	            // ss_SequencialID character string leading zeros addition
	            IF (#si_StringLen < 6)
	            THEN
	                FOR #si_LenFillLoop := 1 TO 6 - #si_StringLen DO
	                    #ss_SequencialID := CONCAT(IN1 := '0',
	                                               IN2 := #ss_SequencialID);
	                END_FOR;
	            END_IF;
	        END_REGION

	        REGION 3.2 LLC Syatem ID
	            // Build LLC Syatem ID
	            #ss_LLCSystemID := CONCAT(IN1 := #is_DEPCOD,
	                                      IN2 := #is_LOConEquipment,
	                                      IN3 := #is_TYPofEquipment,
	                                      IN4 := #is_NumberOfTheEquipment);

	        END_REGION

	        REGION 3.3 - Package ID
	            // Build Package ID
	            #ss_PackageID := CONCAT(IN1 := #is_TrayCellNumber,
	                                    IN2 := #is_SorterNumber,
	                                    IN3 := #is_InductionNumber,
	                                    IN4 := #is_AreaNumber,
	                                    IN5 := #ss_SequencialID);
	        END_REGION

	        REGION 3.4 - Gap

	            // Gap character string clearing
	            #ss_Gap := '';

	            IF ("DB_GIN".GIN[#ii_Gin].General.LeadingGap > 999)
	            THEN
	                #ss_Gap := '999';
	            ELSE

	                // Gap integer input conversion to a character string
	                VAL_STRG(IN := "DB_GIN".GIN[#ii_Gin].General.LeadingGap,
	                         SIZE := 0,
	                         PREC := 0,
	                         FORMAT := 0,
	                         P := 1,
	                         OUT => #ss_Gap);
	                // Length of the gap character string
	                #si_StringLen := LEN(#ss_Gap);
	                // Gap character string leading zeros addition
	                IF (#si_StringLen < 3)
	                THEN
	                    FOR #si_LenFillLoop := 1 TO 3 - #si_StringLen DO
	                        #ss_Gap := CONCAT(IN1 := '0',
	                                          IN2 := #ss_Gap);
	                    END_FOR;
	                END_IF;

	            END_IF;

	        END_REGION

	        REGION 3.5 – Message preparation

	            // Message composing according to the structure: STX,message body,ETX
	            #ss_MessageP1 := CONCAT(IN1 := #cc_STX,
	                                    IN2 := #cs_Length,
	                                    IN3 := #cs_MessageType,
	                                    IN4 := #ss_LLCSystemID,
	                                    IN5 := "DB_GIN".GIN[#ii_Gin].FedEx.ADCSystemID,
	                                    IN6 := "DB_GIN".GIN[#ii_Gin].FedEx.ImageID,
	                                    IN7 := #ss_PackageID,
	                                    IN8 := "DB_GIN".GIN[#ii_Gin].FedEx.HLCPackageID,
	                                    IN9 := "DB_GIN".GIN[#ii_Gin].FedEx.DIMSystemID,
	                                    IN10 := "DB_GIN".GIN[#ii_Gin].FedEx.DIMStatus,
	                                    IN11 := "DB_GIN".GIN[#ii_Gin].FedEx.PackageDimLength,
	                                    IN12 := "DB_GIN".GIN[#ii_Gin].FedEx.PackageDimWidth,
	                                    IN13 := "DB_GIN".GIN[#ii_Gin].FedEx.PackageDimHeight,
	                                    IN14 := #ss_Gap,
	                                    IN15 := "DB_GIN".GIN[#ii_Gin].FedEx.DIMUOM,
	                                    IN16 := "DB_GIN".GIN[#ii_Gin].FedEx.DimLFTstatusCode,
	                                    IN17 := "DB_GIN".GIN[#ii_Gin].FedEx.AlibiDims,
	                                    IN18 := "DB_GIN".GIN[#ii_Gin].FedEx.SCLSystemID,
	                                    IN19 := "DB_GIN".GIN[#ii_Gin].FedEx.SCLWT,
	                                    IN20 := "DB_GIN".GIN[#ii_Gin].FedEx.SCLWTUOM,
	                                    IN21 := "DB_GIN".GIN[#ii_Gin].FedEx.SCLLFTStatusCode,
	                                    IN22 := "DB_GIN".GIN[#ii_Gin].FedEx.AlibiWeight,
	                                    IN23 := "DB_GIN".GIN[#ii_Gin].FedEx.ReasonCode,
	                                    IN24 := "DB_Time".Timestamp,
	                                    IN25 := #iUDT_Facility.TimeZoneDesignator);

	            #ss_MessageP2 := CONCAT(IN1 := "DB_GIN".GIN[#ii_Gin].FedEx.Barcode1Identification,
	                                    IN2 := "DB_GIN".GIN[#ii_Gin].FedEx.Barcode1status,
	                                    IN3 := "DB_GIN".GIN[#ii_Gin].FedEx.Barcode1datalength,
	                                    IN4 := "DB_GIN".GIN[#ii_Gin].FedEx.Barcode1data,
	                                    IN5 := #cc_ETX);

	        END_REGION

	        REGION 3.6 – Maximum number of the message characters

	            #si_MaxMsgLen := "FC_GetNrOfArrayEl"(iv_Array := #sUDT_MessageArray.Character);

	        END_REGION

	        REGION 3.7 – Length of the complete message

	            #si_MsgLen := LEN(#ss_MessageP1) + LEN(#ss_MessageP2);
	            // Message length validation
	            #sa_Status.InvalidMessageLength := #si_MsgLen - 2 <> STRING_TO_INT(#cs_Length);

	        END_REGION

	        REGION 3.8 –  Message array size validation

	            #sa_Status.InvalidMsgArraySize := #si_MsgLen > #si_MaxMsgLen;

	        END_REGION

	        REGION 3.9 –  Message character string conversion to a message array of characters

	            IF (NOT #sa_Status.InvalidMsgArraySize)     // Message character array size is valid
	            THEN

	                Strg_TO_Chars(Strg := #ss_MessageP1,
	                              pChars := 0,
	                              Cnt => #sui_ArrayOffset,
	                              Chars := #sUDT_MessageArray.Character);

	                Strg_TO_Chars(Strg := #ss_MessageP2,
	                              pChars := #sui_ArrayOffset,
	                              Cnt => #sui_MsgArrayElNr,
	                              Chars := #sUDT_MessageArray.Character);

	            END_IF;

	        END_REGION

	        REGION 3.10 – Clearing remaining characters in the message character array

	            IF (NOT #sa_Status.InvalidMsgArraySize)     // Message character array size is valid
	            THEN

	                // Filling up not used message character array elements with '$00' (ASCII - 16#00)
	                FILL_BLK(IN := #cc_NULL,                                                                             // Fill not used message char array elements with '$00'
	                         COUNT := UINT_TO_ULINT(INT_TO_UINT(#si_MaxMsgLen) - #sui_MsgArrayElNr - #sui_ArrayOffset),
	                         OUT => #sUDT_MessageArray.Character[#sui_MsgArrayElNr + #sui_ArrayOffset]);

	            END_IF;

	        END_REGION

	        REGION 3.11 – Message write into a FIFO register

	            IF NOT #sa_Status.InvalidMsgArraySize               // Message character array size is valid
	                AND NOT #sa_Status.InvalidMessageLength         //Message length is valid
	            THEN

	                // Mode 'W' - Write FIFO record
	                "FC_Fifo"(ic_Mode := 'W',
	                          qUDT_Status => #sa_Status.FIFOStatus,
	                          qx_Error => #sa_Status.FIFOError,
	                          qx_Warning => #sa_Status.FIFOWarning,
	                          iqv_Data := #sUDT_MessageArray,
	                          iqUDT_FifoHeader := #iqUDT_FifoHeader,
	                          iqv_DataBuffer := #iqa_FifoData);
	            ELSE
	                // Increase counter messages not sent because of wrong message length
	                #sa_Statistics.NotSentWrongMsgLen += 1;

	            END_IF;

	            #si_OldGin := #ii_Gin;
	        END_REGION


	        // In case of FIFO full, the FIFO full error bit and FIFO collective error bit are set
	    ELSE
	        #sa_Status.FIFOError := TRUE;
	        #sa_Status.FIFOStatus.FifoFull := TRUE;
	    END_IF;



	END_REGION

	REGION 4 - Writing outputs

	    #sx_Error := #sa_Status.InvalidMessageLength        // Invalid message length
	    OR #sa_Status.InvalidGIN                            // Invalid GIN
	    OR #sa_Status.InvalidMsgArraySize                   // Invalid message array size
	    OR #sa_Status.FIFOError;                            // FIFO error

	END_REGION



	REGION 5 Unexpected DX Request

	    IF #iqx_Unexpected_DX_Req THEN

	        REGION 5.1 – FIFO header status update

	            // Mode 'S' - FIFO register status update
	            "FC_Fifo"(ic_Mode := 'S',
	                      qUDT_Status => #sa_Status.FIFOStatus,
	                      qx_Error => #sa_Status.FIFOError,
	                      qx_Warning => #sa_Status.FIFOWarning,
	                      iqv_Data := #sUDT_MessageArray,
	                      iqUDT_FifoHeader := #iqUDT_FifoHeader,
	                      iqv_DataBuffer := #iqa_FifoData);
	        END_REGION

	        REGION 5.2 – Message preparation

	            IF NOT #iqUDT_FifoHeader.Status.Full       // FIFO isn't full
	            THEN
	                REGION Sequencial ID
	                    // ss_SequencialID character string clearing
	                    #ss_SequencialID := '';
	                    // ss_SequencialID integer input conversion to a character string
	                    VAL_STRG(IN := "DB_ExternalGIN".UnexpectedSI.FedEx.CustomerID,
	                             SIZE := 0,
	                             PREC := 0,
	                             FORMAT := 0,
	                             P := 1,
	                             OUT => #ss_SequencialID);
	                    // Length of the ss_SequencialID character string
	                    #si_StringLen := LEN(#ss_SequencialID);

	                    // ss_SequencialID character string leading zeros addition
	                    IF (#si_StringLen < 6)
	                    THEN
	                        FOR #si_LenFillLoop := 1 TO 6 - #si_StringLen DO
	                            #ss_SequencialID := CONCAT(IN1 := '0',
	                                                       IN2 := #ss_SequencialID);
	                        END_FOR;
	                    END_IF;
	                END_REGION

	                REGION LLC Syatem ID
	                    // Build LLC Syatem ID
	                    #ss_LLCSystemID := CONCAT(IN1 := #is_DEPCOD,
	                                              IN2 := #is_LOConEquipment,
	                                              IN3 := #is_TYPofEquipment,
	                                              IN4 := #is_NumberOfTheEquipment);

	                END_REGION

	                REGION Package ID
	                    // Build Package ID
	                    #ss_PackageID := CONCAT(IN1 := #is_TrayCellNumber,
	                                            IN2 := #is_SorterNumber,
	                                            IN3 := #is_InductionNumber,
	                                            IN4 := #is_AreaNumber,
	                                            IN5 := #ss_SequencialID);
	                END_REGION

	                REGION Gap

	                    #ss_Gap := '000';

	                END_REGION

	                REGION 3.5 – Message preparation

	                    // Message composing according to the structure: STX,message body,ETX
	                    #ss_MessageP1 := CONCAT(IN1 := #cc_STX,
	                                            IN2 := #cs_Length,
	                                            IN3 := #cs_MessageType,
	                                            IN4 := #ss_LLCSystemID,
	                                            IN5 := "DB_ExternalGIN".UnexpectedSI.FedEx.ADCSystemID,
	                                            IN6 := "DB_ExternalGIN".UnexpectedSI.FedEx.ImageID,
	                                            IN7 := "DB_ExternalGIN".UnexpectedSI.FedEx.PackageID,
	                                            IN8 := "DB_ExternalGIN".UnexpectedSI.FedEx.HLCPackageID,
	                                            IN9 := "DB_ExternalGIN".UnexpectedSI.FedEx.DIMSystemID,
	                                            IN10 := "DB_ExternalGIN".UnexpectedSI.FedEx.DIMStatus,
	                                            IN11 := "DB_ExternalGIN".UnexpectedSI.FedEx.PackageDimLength,
	                                            IN12 := "DB_ExternalGIN".UnexpectedSI.FedEx.PackageDimWidth,
	                                            IN13 := "DB_ExternalGIN".UnexpectedSI.FedEx.PackageDimHeight,
	                                            IN14 := #ss_Gap,
	                                            IN15 := "DB_ExternalGIN".UnexpectedSI.FedEx.DIMUOM,
	                                            IN16 := "DB_ExternalGIN".UnexpectedSI.FedEx.DimLFTstatusCode,
	                                            IN17 := "DB_ExternalGIN".UnexpectedSI.FedEx.AlibiDims,
	                                            IN18 := "DB_ExternalGIN".UnexpectedSI.FedEx.SCLSystemID,
	                                            IN19 := "DB_ExternalGIN".UnexpectedSI.FedEx.SCLWT,
	                                            IN20 := "DB_ExternalGIN".UnexpectedSI.FedEx.SCLWTUOM,
	                                            IN21 := "DB_ExternalGIN".UnexpectedSI.FedEx.SCLLFTStatusCode,
	                                            IN22 := "DB_ExternalGIN".UnexpectedSI.FedEx.AlibiWeight,
	                                            IN23 := "DB_ExternalGIN".UnexpectedSI.FedEx.ReasonCode,
	                                            IN24 := "DB_Time".Timestamp,
	                                            IN25 := #iUDT_Facility.TimeZoneDesignator);

	                    #ss_MessageP2 := CONCAT(IN1 := "DB_ExternalGIN".UnexpectedSI.FedEx.Barcode1Identification,
	                                            IN2 := "DB_ExternalGIN".UnexpectedSI.FedEx.Barcode1status,
	                                            IN3 := "DB_ExternalGIN".UnexpectedSI.FedEx.Barcode1datalength,
	                                            IN4 := "DB_ExternalGIN".UnexpectedSI.FedEx.Barcode1data,
	                                            IN5 := #cc_ETX);

	                END_REGION

	                REGION 3.6 – Maximum number of the message characters

	                    #si_MaxMsgLen := "FC_GetNrOfArrayEl"(iv_Array := #sUDT_MessageArray.Character);

	                END_REGION

	                REGION 3.7 – Length of the complete message

	                    #si_MsgLen := LEN(#ss_MessageP1) + LEN(#ss_MessageP2);
	                    // Message length validation
	                    #sa_Status.InvalidMessageLength := #si_MsgLen - 2 <> STRING_TO_INT(#cs_Length);

	                END_REGION

	                REGION 3.8 –  Message array size validation

	                    #sa_Status.InvalidMsgArraySize := #si_MsgLen > #si_MaxMsgLen;

	                END_REGION

	                REGION 3.9 –  Message character string conversion to a message array of characters

	                    IF (NOT #sa_Status.InvalidMsgArraySize)     // Message character array size is valid
	                    THEN

	                        Strg_TO_Chars(Strg := #ss_MessageP1,
	                                      pChars := 0,
	                                      Cnt => #sui_ArrayOffset,
	                                      Chars := #sUDT_MessageArray.Character);

	                        Strg_TO_Chars(Strg := #ss_MessageP2,
	                                      pChars := #sui_ArrayOffset,
	                                      Cnt => #sui_MsgArrayElNr,
	                                      Chars := #sUDT_MessageArray.Character);

	                    END_IF;

	                END_REGION

	                REGION 3.10 – Clearing remaining characters in the message character array

	                    IF (NOT #sa_Status.InvalidMsgArraySize)     // Message character array size is valid
	                    THEN

	                        // Filling up not used message character array elements with '$00' (ASCII - 16#00)
	                        FILL_BLK(IN := #cc_NULL,                                                                             // Fill not used message char array elements with '$00'
	                                 COUNT := UINT_TO_ULINT(INT_TO_UINT(#si_MaxMsgLen) - #sui_MsgArrayElNr - #sui_ArrayOffset),
	                                 OUT => #sUDT_MessageArray.Character[#sui_MsgArrayElNr + #sui_ArrayOffset]);

	                    END_IF;

	                END_REGION

	                REGION 3.11 – Message write into a FIFO register

	                    IF NOT #sa_Status.InvalidMsgArraySize               // Message character array size is valid
	                        AND NOT #sa_Status.InvalidMessageLength         //Message length is valid
	                    THEN

	                        // Mode 'W' - Write FIFO record
	                        "FC_Fifo"(ic_Mode := 'W',
	                                  qUDT_Status => #sa_Status.FIFOStatus,
	                                  qx_Error => #sa_Status.FIFOError,
	                                  qx_Warning => #sa_Status.FIFOWarning,
	                                  iqv_Data := #sUDT_MessageArray,
	                                  iqUDT_FifoHeader := #iqUDT_FifoHeader,
	                                  iqv_DataBuffer := #iqa_FifoData);
	                    ELSE
	                        // Increase counter messages not sent because of wrong message length
	                        #sa_Statistics.NotSentWrongMsgLen += 1;

	                    END_IF;

	                END_REGION
	                #iqx_Unexpected_DX_Req := FALSE;


	                // In case of FIFO full, the FIFO full error bit and FIFO collective error bit are set
	            ELSE
	                #sa_Status.FIFOError := TRUE;
	                #sa_Status.FIFOStatus.FifoFull := TRUE;
	            END_IF;

	        END_REGION
	    END_IF;
	END_REGION



	REGION 6 - Writing outputs

	    #qx_Error := #sa_Status.InvalidMessageLength        // Invalid message length
	    OR #sa_Status.InvalidGIN                            // Invalid GIN
	    OR #sa_Status.InvalidMsgArraySize                   // Invalid message array size
	    OR #sa_Status.FIFOError                             // FIFO error
	    OR #sx_Error;

	END_REGION
END_FUNCTION_BLOCK

FUNCTION_BLOCK "FB_FedExEntrancePoint"
{ S7_Optimized_Access := 'TRUE' }
VERSION : 0.1
// ATTRIBUTES
// AUTO_NUMBER = True
// BLOCK_NUMBER = 71
// END_ATTRIBUTES
   VAR_INPUT
      is_PackageEntrancePoint { ExternalAccessible := 'False'; ExternalVisible := 'False'; ExternalWritable := 'False'} : String;
      is_PackageEntranceState { ExternalAccessible := 'False'; ExternalVisible := 'False'; ExternalWritable := 'False'} : String;
      ii_Gin { ExternalAccessible := 'False'; ExternalVisible := 'False'; ExternalWritable := 'False'} : Int;
   END_VAR

   VAR
      si_OldGIN { ExternalAccessible := 'False'; ExternalVisible := 'False'; ExternalWritable := 'False'} : Int;
      si_StringLen { ExternalAccessible := 'False'; ExternalVisible := 'False'; ExternalWritable := 'False'} : Int;
      si_LenFillLoop { ExternalAccessible := 'False'; ExternalVisible := 'False'; ExternalWritable := 'False'} : Int;
   END_VAR

   VAR_TEMP
      tx_InvalidGIN : Bool;
   END_VAR


BEGIN
	(*
	----------------------------------------------------------------------------------------

	Version history:
	Date        | Version   | Author        | Remark
	----------------------------------------------------------------------------------------
	30/06/2022  | 0.1       | K. Pokorski   | first release MHS TIA 16
	21/02/2023  | 4.0       | F.Baten       | 4.0 Release TIA 17.5
	*)

	REGION 1 - GIN validation

	    // GIN validation
	    #tx_InvalidGIN := (#ii_Gin < 1) OR (#ii_Gin > 9999);

	    IF #ii_Gin <> #si_OldGIN AND NOT #tx_InvalidGIN
	    THEN

	        "DB_GIN".GIN[#ii_Gin].FedEx.PackageEntrancePoint := #is_PackageEntrancePoint;
	        "DB_GIN".GIN[#ii_Gin].FedEx.PackageEntranceState := #is_PackageEntranceState;

	        #si_StringLen := LEN("DB_GIN".GIN[#ii_Gin].FedEx.PackageEntrancePoint);

	        IF (#si_StringLen < 14)
	        THEN
	            FOR #si_LenFillLoop := 1 TO 14 - #si_StringLen DO

	                "DB_GIN".GIN[#ii_Gin].FedEx.PackageEntrancePoint := CONCAT(IN1 := "DB_GIN".GIN[#ii_Gin].FedEx.PackageEntrancePoint,
	                                                                           IN2 := ' ');
	            END_FOR;
	        END_IF;

	        #si_OldGIN := #ii_Gin;

	    END_IF;


	END_REGION






END_FUNCTION_BLOCK

FUNCTION_BLOCK "FB_FedExGetPositionPolisorter"
TITLE = FB_GetPosition
{ S7_Optimized_Access := 'TRUE' }
FAMILY : MHS
VERSION : 3.0
// ATTRIBUTES
// AUTO_NUMBER = True
// BLOCK_NUMBER = 73
// END_ATTRIBUTES
//Function to find the position based on the GIN in the tracking.
   VAR_INPUT
      idi_ConveyorLength { ExternalAccessible := 'False'; ExternalVisible := 'False'; ExternalWritable := 'False'} : DInt;   // Conveyor length [mm]
      idi_WaitDistanceCorrection { ExternalAccessible := 'False'; ExternalVisible := 'False'; ExternalWritable := 'False'} : DInt := 10000;   // Distance how much parcel tail can stick out of the conveyor [mm]
   END_VAR

   VAR_IN_OUT
      iqs_DBDestination : Array[*] of "UDT_FedExDestinations";   // Array with destination data for parcel
      iqUDT_PolisorterInterface : "UDT_PolisorterInterface";   // Interface beween VSU and VFD
      iqUDT_ConveyorInterface : "UDT_ConveyorInterface";   // Polisorter conveyor interface structure
      iqs_TrackingData : Array[*] of Int;   // Tracking data
   END_VAR

   VAR
      si_Gin { ExternalAccessible := 'False'; ExternalVisible := 'False'; ExternalWritable := 'False'} : Int;   // GIN
      si_PreviousGin { ExternalAccessible := 'False'; ExternalVisible := 'False'; ExternalWritable := 'False'} : Int;   // Old GIN memeory
      si_RequestedDestination { ExternalAccessible := 'False'; ExternalVisible := 'False'; ExternalWritable := 'False'} : Int;   // The destination for this GIN
      si_RequestedPosition { ExternalAccessible := 'False'; ExternalVisible := 'False'; ExternalWritable := 'False'} : Int;   // Requested position
      si_LC_Positions { ExternalAccessible := 'False'; ExternalVisible := 'False'; ExternalWritable := 'False'} : Int;   // Loopcounter positions
      si_LC_Destinations { ExternalAccessible := 'False'; ExternalVisible := 'False'; ExternalWritable := 'False'} : Int;   // Loopcounter destinations
      si_NrPositons { ExternalAccessible := 'False'; ExternalVisible := 'False'; ExternalWritable := 'False'} : Int;   // Number of positions in the search area
      si_NrDestinations { ExternalAccessible := 'False'; ExternalVisible := 'False'; ExternalWritable := 'False'} : Int;   // Number of destinations per position
      sx_NewGinFound { ExternalAccessible := 'False'; ExternalVisible := 'False'; ExternalWritable := 'False'} : Bool;   // Memory to start searching
      sdi_WaitDistance { ExternalAccessible := 'False'; ExternalVisible := 'False'; ExternalWritable := 'False'} : DInt;   // Calculated wait distance [cm]
      sdi_ParcelLength { ExternalAccessible := 'False'; ExternalVisible := 'False'; ExternalWritable := 'False'} : DInt;   // Parcel length [cm]
   END_VAR


BEGIN
	(*
	----------------------------------------------------------------------------------------
	|                                                                                      |
	|  Copyright  2019             MHS                                                     |
	|  All Rights Reserved         Larenweg 90                                             |
	|                              5234 KC 's-Hertogenbosch,                               |
	|                              Netherlands                                             |
	|                                                                                      |
	----------------------------------------------------------------------------------------

	Version history:
	Date        | Version   | Author        | Remark
	----------------------------------------------------------------------------------------

	26/01/2022  | 0.1       | L.Klar        | Initial version
	13/03/2024  | 4.1       | S. Nieświec   | 4.1 Release TIA 18
	02/05/2024  | 4.2       | J.Majer      | Datatype conversions changed from automatic to explicit, to accomodate IEC 61131-3 standard
	*)

	REGION 1 - Determine size of search area

	    #si_NrPositons := "FC_GetNrOfArrayEl"(#iqs_DBDestination);
	    #si_NrDestinations := "FC_GetNrOfArrayEl"(#iqs_DBDestination[1].Destination);

	END_REGION

	REGION 2 - Get GIN from tracking DB

	    // There is a value in the tracking data on the decision point which is not '0' or equal to the previous GIN
	    IF (#iqs_TrackingData[#iqUDT_PolisorterInterface.Decisionpoint] <> 0) AND (#iqs_TrackingData[#iqUDT_PolisorterInterface.Decisionpoint] <> #si_PreviousGin)
	    THEN
	        #si_Gin := #iqs_TrackingData[#iqUDT_PolisorterInterface.Decisionpoint];
	        #sx_NewGinFound := TRUE;
	    END_IF;

	END_REGION

	REGION 3 - Wait distance

	    IF #sdi_WaitDistance > 0 THEN
	        #sdi_WaitDistance -= #iqUDT_ConveyorInterface.Displacement;
	    END_IF;

	END_REGION

	REGION 4 - Get destination from GIN DB
	    // If new GIN has been detected, get destination from its GIN record

	    IF #sx_NewGinFound AND #si_Gin > 0
	    THEN
	        #si_RequestedDestination := DINT_TO_INT("DB_GIN".GIN[#si_Gin].General.Destination[0]);

	        #sdi_ParcelLength := "DB_GIN".GIN[#si_Gin].General.Length;

	        // If parcel length is lower than conveyor length - decision point use calculated decision point to switch.
	        // If not, then caluclate additional wait distance, based on correction factor
	        // If the parcel length is equal to 0, use fixed wait distance of decision point minus 40
	        IF #sdi_ParcelLength > 0
	        THEN
	            IF #sdi_ParcelLength < #idi_ConveyorLength / 10 - #iqUDT_PolisorterInterface.Decisionpoint
	            THEN
	                #sdi_WaitDistance := 0;
	            ELSE
	                #sdi_WaitDistance := #sdi_ParcelLength - (#idi_ConveyorLength / 10 - #iqUDT_PolisorterInterface.Decisionpoint) - #idi_WaitDistanceCorrection / 10;
	            END_IF;
	        ELSE
	            #sdi_WaitDistance := #iqUDT_PolisorterInterface.Decisionpoint - 40;
	        END_IF;
	        #si_PreviousGin := #si_Gin;
	        #si_Gin := 0;
	        #iqUDT_PolisorterInterface.RequestedPosition := 0;

	    END_IF;

	END_REGION

	REGION 5 - Get requested position when new GIN is found

	    IF #sx_NewGinFound AND #sdi_WaitDistance <= 0
	    THEN
	        // If destination is different than 0, find a position in destination arrays. Otherwise, requested position is set to default.
	        IF #si_RequestedDestination <> 0 THEN
	            FOR #si_LC_Positions := 1 TO #si_NrPositons BY 1 DO
	                FOR #si_LC_Destinations := 0 TO (#si_NrDestinations - 1) BY 1 DO
	                    IF #iqs_DBDestination[#si_LC_Positions].Destination[#si_LC_Destinations] = #si_RequestedDestination
	                    THEN
	                        #si_RequestedPosition := #si_LC_Positions;
	                        EXIT;
	                    END_IF;
	                END_FOR;
	                // Position found
	                IF #si_RequestedPosition <> 0
	                THEN
	                    #iqUDT_PolisorterInterface.RequestedPosition := #si_RequestedPosition;
	                    #sx_NewGinFound := FALSE;
	                    #si_RequestedPosition := 0;
	                    EXIT;
	                END_IF;
	            END_FOR;
	        ELSE
	            // Default position
	            #sx_NewGinFound := FALSE;
	            #iqUDT_PolisorterInterface.RequestedPosition := 99;
	            #si_RequestedPosition := 0;
	        END_IF;
	    END_IF;
	END_REGION
END_FUNCTION_BLOCK

FUNCTION_BLOCK "FB_FedExInsertPoint"
{ S7_Optimized_Access := 'TRUE' }
VERSION : 0.1
// ATTRIBUTES
// AUTO_NUMBER = True
// BLOCK_NUMBER = 75
// END_ATTRIBUTES
   VAR_INPUT
      iUDT_ConveyorCommonConfiguration { ExternalAccessible := 'False'; ExternalVisible := 'False'; ExternalWritable := 'False'} : "UDT_ConveyorCommonConfiguration";   // Common configuration of insert conveyor
      iUDT_ConveyorInterface { ExternalAccessible := 'False'; ExternalVisible := 'False'; ExternalWritable := 'False'} : "UDT_ConveyorInterface";   // Insert conveyor interface
      idi_EoSPosition { ExternalAccessible := 'False'; ExternalVisible := 'False'; ExternalWritable := 'False'} : DInt;   // End of section sensor position [mm]
      ix_KeySwitch { ExternalAccessible := 'False'; ExternalVisible := 'False'; ExternalWritable := 'False'} : Bool;   // TRUE when insert mode active
      ix_PushButton { ExternalAccessible := 'False'; ExternalVisible := 'False'; ExternalWritable := 'False'} : Bool;   // TRUE when push button pressed
      ix_InsertConveyorEoS { ExternalAccessible := 'False'; ExternalVisible := 'False'; ExternalWritable := 'False'} : Bool;   // End of section sensor of insert conveyor
   END_VAR

   VAR_OUTPUT
      qx_UpstreamConveyorHold { ExternalAccessible := 'False'; ExternalVisible := 'False'; ExternalWritable := 'False'} : Bool;   // Hold insert's upstream conveyor
      qx_InsertConveyorHold { ExternalAccessible := 'False'; ExternalVisible := 'False'; ExternalWritable := 'False'} : Bool;   // Hold insert conveyor
      qx_Indicator { ExternalAccessible := 'False'; ExternalVisible := 'False'; ExternalWritable := 'False'} : Bool;   // Blue lamp on push button
      qx_InsertModeActive { ExternalAccessible := 'False'; ExternalVisible := 'False'; ExternalWritable := 'False'} : Bool;
   END_VAR

   VAR
      sR_TRIG_ModeChange {InstructionName := 'R_TRIG'; LibVersion := '1.0'; ExternalAccessible := 'False'; ExternalVisible := 'False'; ExternalWritable := 'False'; S7_SetPoint := 'False'} : R_TRIG;   // Mode change detection
      sR_TRIG_InsertMode {InstructionName := 'R_TRIG'; LibVersion := '1.0'; ExternalAccessible := 'False'; ExternalVisible := 'False'; ExternalWritable := 'False'; S7_SetPoint := 'False'} : R_TRIG;   // Insert mode activation
      sF_TRIG_FlowMode {InstructionName := 'F_TRIG'; LibVersion := '1.0'; ExternalAccessible := 'False'; ExternalVisible := 'False'; ExternalWritable := 'False'; S7_SetPoint := 'False'} : F_TRIG;   // Flow mode activation
      sR_TRIG_PushButton {InstructionName := 'R_TRIG'; LibVersion := '1.0'; ExternalAccessible := 'False'; ExternalVisible := 'False'; ExternalWritable := 'False'; S7_SetPoint := 'False'} : R_TRIG;   // Push button trigger
      sR_TRIG_EoS {InstructionName := 'R_TRIG'; LibVersion := '1.0'; ExternalAccessible := 'False'; ExternalVisible := 'False'; ExternalWritable := 'False'; S7_SetPoint := 'False'} : R_TRIG;   // End of section sensor trigger
      si_DistanceToStop { ExternalAccessible := 'False'; ExternalVisible := 'False'; ExternalWritable := 'False'} : DInt;   // Distance from end conveyor to stop [cm]
      sx_ClearingSequence { ExternalAccessible := 'False'; ExternalVisible := 'False'; ExternalWritable := 'False'} : Bool;   // Clearing sequence active
      sx_ReleaseSequence { ExternalAccessible := 'False'; ExternalVisible := 'False'; ExternalWritable := 'False'} : Bool;   // Release sequence active
      sx_ParcelPositionCorrectMode { ExternalAccessible := 'False'; ExternalVisible := 'False'; ExternalWritable := 'False'} : Bool;   // Position correction active
      sx_InsertModeActive { ExternalAccessible := 'False'; ExternalVisible := 'False'; ExternalWritable := 'False'} : Bool;
   END_VAR


BEGIN
	(*
	----------------------------------------------------------------------------------------

	Version history:
	Date        | Version   | Author        | Remark
	----------------------------------------------------------------------------------------
	18/03/2022  | 1.0       | K.Pokorski    | first release MHS TIA 16
	28/06/2022  | 1.1       | K.Pokorski    | Adjust software for monostable key
	21/02/2023  | 4.0       | F.Baten       | 4.0 Release TIA 17.5
	*)


	REGION 1 - Change Mode detection

	    #sR_TRIG_ModeChange(CLK := #ix_KeySwitch);

	    IF #sR_TRIG_ModeChange.Q
	    THEN
	        IF #sx_InsertModeActive THEN
	            #sx_InsertModeActive := FALSE;
	        ELSE
	            #sx_InsertModeActive := TRUE;
	        END_IF;
	    END_IF;

	    #sR_TRIG_InsertMode(CLK := #sx_InsertModeActive);

	    #sF_TRIG_FlowMode(CLK := #sx_InsertModeActive);

	    #sR_TRIG_PushButton(CLK := #ix_PushButton);

	    #sR_TRIG_EoS(CLK := #ix_InsertConveyorEoS);


	END_REGION

	REGION 2 - Insert mode

	    // Key switch in insert mode
	    IF #sx_InsertModeActive THEN

	        // Enable clearing sequence
	        IF #sR_TRIG_InsertMode.Q THEN
	            #si_DistanceToStop := #iUDT_ConveyorCommonConfiguration.Length / 10;
	            #qx_UpstreamConveyorHold := TRUE;
	            #sx_ClearingSequence := TRUE;
	            #sx_ReleaseSequence := FALSE;
	        END_IF;

	        // Indicator control
	        IF #sx_ClearingSequence THEN
	            #qx_Indicator := TRUE;
	        ELSE
	            #qx_Indicator := "DB_Memory".Clock_1Hz;
	        END_IF;

	        // Clearing sequence control
	        IF #sx_ClearingSequence THEN
	            #si_DistanceToStop -= #iUDT_ConveyorInterface.Displacement;
	            IF #si_DistanceToStop <= 0 THEN
	                #qx_InsertConveyorHold := TRUE;
	                #sx_ClearingSequence := FALSE;
	            ELSE
	                #qx_InsertConveyorHold := FALSE;
	            END_IF;
	        END_IF;

	        // Enable release sequence
	        IF #sR_TRIG_PushButton.Q AND NOT #sx_ClearingSequence THEN
	            #sx_ReleaseSequence := TRUE;
	            #si_DistanceToStop := (#iUDT_ConveyorCommonConfiguration.Length / 10);
	        END_IF;

	        // Release sequence control
	        IF #sx_ReleaseSequence THEN

	            IF #sR_TRIG_EoS.Q THEN
	                #si_DistanceToStop := #idi_EoSPosition / 10;
	            END_IF;

	            #si_DistanceToStop -= #iUDT_ConveyorInterface.Displacement;

	            IF #si_DistanceToStop <= 0 THEN
	                #qx_InsertConveyorHold := TRUE;
	                #sx_ReleaseSequence := FALSE;
	            ELSE
	                #qx_InsertConveyorHold := FALSE;
	            END_IF;

	        END_IF;

	    END_IF;

	    #qx_InsertModeActive := #sx_InsertModeActive;

	END_REGION


	REGION 3 - Flow Mode

	    // Key switch in flow mode
	    IF NOT #sx_InsertModeActive THEN

	        // Initialize flow mode
	        IF #sF_TRIG_FlowMode.Q THEN

	            #qx_InsertConveyorHold := FALSE;
	            #qx_UpstreamConveyorHold := FALSE;
	            #sx_ParcelPositionCorrectMode := FALSE;

	        END_IF;

	        // Position correct mode enable
	        IF #sR_TRIG_PushButton.Q AND NOT #sx_ParcelPositionCorrectMode THEN

	            #qx_InsertConveyorHold := TRUE;
	            #sx_ParcelPositionCorrectMode := TRUE;

	            // Position correct mode disable
	        ELSIF #sR_TRIG_PushButton.Q AND #sx_ParcelPositionCorrectMode THEN

	            #qx_InsertConveyorHold := FALSE;
	            #sx_ParcelPositionCorrectMode := FALSE;

	        END_IF;

	        // Indicator control
	        #qx_Indicator := "DB_Memory".Clock_1Hz AND #sx_ParcelPositionCorrectMode;

	    END_IF;
	END_REGION
END_FUNCTION_BLOCK

FUNCTION_BLOCK "FB_FedExTriggerEventMessage"
TITLE = FB_Heartbeat
{ S7_Optimized_Access := 'TRUE' }
AUTHOR : MHSE
FAMILY : UPS_SpecificCommunication
VERSION : 3.0
// ATTRIBUTES
// AUTO_NUMBER = True
// BLOCK_NUMBER = 85
// END_ATTRIBUTES
//Function block to send and monitor the UPS heartbeat message.
   VAR_INPUT
      iUDT_Facility { ExternalAccessible := 'False'; ExternalVisible := 'False'; ExternalWritable := 'False'} : "UDT_FedExFacility";   // System configuration
      is_LOConEquipment { ExternalAccessible := 'False'; ExternalVisible := 'False'; ExternalWritable := 'False'} : String[3];   // Location of the equipment
      is_DEPCOD { ExternalAccessible := 'False'; ExternalVisible := 'False'; ExternalWritable := 'False'} : String[6];   // Depot Code
      is_TYPofEquipment { ExternalAccessible := 'False'; ExternalVisible := 'False'; ExternalWritable := 'False'} : String[3];   // Type of equipment
      is_NumberOfTheEquipment { ExternalAccessible := 'False'; ExternalVisible := 'False'; ExternalWritable := 'False'} : String[3];   // Number of the equipment 001-999
      is_TrayCellNumber { ExternalAccessible := 'False'; ExternalVisible := 'False'; ExternalWritable := 'False'} : String[3];   // Tray/Cell number (for loop sorters) or generated by LLC (on line sorters).
      is_SorterNumber { ExternalAccessible := 'False'; ExternalVisible := 'False'; ExternalWritable := 'False'} : String[2];   // Sorter number
      is_InductionNumber { ExternalAccessible := 'False'; ExternalVisible := 'False'; ExternalWritable := 'False'} : String[2];   // Induction number
      is_AreaNumber { ExternalAccessible := 'False'; ExternalVisible := 'False'; ExternalWritable := 'False'} : String[2];   // Area number
      is_IncompatiblesUnit { ExternalAccessible := 'False'; ExternalVisible := 'False'; ExternalWritable := 'False'} : String[2];   // Id of the unit to be trigger inside the CWC. (e.g Scale1=S1; Scale2=S2).
      ii_Gin { ExternalAccessible := 'False'; ExternalVisible := 'False'; ExternalWritable := 'False'} : Int;   // GIN number
   END_VAR

   VAR_OUTPUT
      qx_Error { ExternalAccessible := 'False'; ExternalVisible := 'False'; ExternalWritable := 'False'} : Bool;   // Error
   END_VAR

   VAR_IN_OUT
      iqUDT_FifoHeader : "UDT_FifoHeader";   // FIFO header
      iqa_FifoData : Array[*] of "UDT_Message";   // FIFO data
   END_VAR

   VAR
      sUDT_MessageArray { ExternalAccessible := 'False'; ExternalVisible := 'False'; ExternalWritable := 'False'; S7_SetPoint := 'False'} : "UDT_Message";   // Message character array
      sa_Status { ExternalAccessible := 'False'; ExternalVisible := 'False'; ExternalWritable := 'False'} : Struct   // Status structure
         FIFOStatus { ExternalAccessible := 'False'; ExternalVisible := 'False'; ExternalWritable := 'False'} : "UDT_FifoStatus";   // FIFO status structure
         FIFOError { ExternalAccessible := 'False'; ExternalVisible := 'False'; ExternalWritable := 'False'; S7_SetPoint := 'True'} : Bool;   // FIFO data buffer full
         FIFOWarning { ExternalAccessible := 'False'; ExternalVisible := 'False'; ExternalWritable := 'False'; S7_SetPoint := 'True'} : Bool;   // FIFO error
         InvalidGIN { ExternalAccessible := 'False'; ExternalVisible := 'False'; ExternalWritable := 'False'} : Bool;   // Invalid GIN
         InvalidMessageLength { ExternalAccessible := 'False'; ExternalVisible := 'False'; ExternalWritable := 'False'} : Bool;   // Calculated message length is different than required
         InvalidMsgArraySize { ExternalAccessible := 'False'; ExternalVisible := 'False'; ExternalWritable := 'False'} : Bool;   // Length of the message is bigger than length of message array
      END_STRUCT;
      sa_Statistics { ExternalAccessible := 'False'; ExternalVisible := 'False'; ExternalWritable := 'False'} : Struct   // Statistics structure
         NotSentWrongMsgLen { ExternalAccessible := 'False'; ExternalVisible := 'False'; ExternalWritable := 'False'} : DInt;   // COMISSIONING PURPOSE Messages not sent because built message length does not match with required message length
      END_STRUCT;
      ss_LLCSystemID { ExternalAccessible := 'False'; ExternalVisible := 'False'; ExternalWritable := 'False'} : String[15];   // Identifier of Low-Level controls
      ss_SequencialID { ExternalAccessible := 'False'; ExternalVisible := 'False'; ExternalWritable := 'False'} : String[6];   // Identifier of Low-Level controls
      ss_Message { ExternalAccessible := 'False'; ExternalVisible := 'False'; ExternalWritable := 'False'} : String;   // Message character string
      ss_PackageID { ExternalAccessible := 'False'; ExternalVisible := 'False'; ExternalWritable := 'False'} : String;   // Identifier of Low-Level controls
      ss_Gap { ExternalAccessible := 'False'; ExternalVisible := 'False'; ExternalWritable := 'False'} : String;   // Parcel leading gap
      ss_GapUOM { ExternalAccessible := 'False'; ExternalVisible := 'False'; ExternalWritable := 'False'} : String;   // Gap units
      sui_MsgArrayElNr { ExternalAccessible := 'False'; ExternalVisible := 'False'; ExternalWritable := 'False'} : UInt;   // Message array size
      si_OldGin { ExternalAccessible := 'False'; ExternalVisible := 'False'; ExternalWritable := 'False'} : Int;   // Previous Gin
      si_StringLen { ExternalAccessible := 'False'; ExternalVisible := 'False'; ExternalWritable := 'False'} : Int;   // Length of string used in loops to pad string with spaces or 0
      si_LenFillLoop { ExternalAccessible := 'False'; ExternalVisible := 'False'; ExternalWritable := 'False'} : Int;   // Loop couter
      si_MaxMsgLen { ExternalAccessible := 'False'; ExternalVisible := 'False'; ExternalWritable := 'False'} : Int;   // Maximum message length
      si_MsgLen { ExternalAccessible := 'False'; ExternalVisible := 'False'; ExternalWritable := 'False'} : Int;   // String character message length
   END_VAR

   VAR CONSTANT
      cc_NULL : Char := '$00';   // NULL sign
      cs_Start : Char := '$02';   // Start of the text
      cs_End : Char := '$03';   // End of the text
      cs_Length : String := '0142';   // Legth of the message
      cs_MessageType : String := 'TE';   // Message type
   END_VAR


BEGIN
	(*
	----------------------------------------------------------------------------------------

	Version history:
	Date        | Version   | Author        | Remark
	----------------------------------------------------------------------------------------
	29/06/2021  | 1.0       | F.Baten       | first release MHS TIA 16.0
	10/11/2021  | 1.2       | M.Piela       | Updating regions numbering
	26/04/2022  | 1.3       | K. Pokorski   | Review
	21/02/2023  | 4.0       | F.Baten       | 4.0 Release TIA 17.5
	*)

	REGION 1 – FIFO header status update

	    // Mode 'S' - FIFO register status update
	    "FC_Fifo"(ic_Mode := 'S',
	              qUDT_Status => #sa_Status.FIFOStatus,
	              qx_Error => #sa_Status.FIFOError,
	              qx_Warning => #sa_Status.FIFOWarning,
	              iqv_Data := #sUDT_MessageArray,
	              iqUDT_FifoHeader := #iqUDT_FifoHeader,
	              iqv_DataBuffer := #iqa_FifoData);
	END_REGION

	REGION GIN validation

	    // GIN validation
	    #sa_Status.InvalidGIN :=
	    #ii_Gin < 1
	    OR #ii_Gin > 9999;
	END_REGION

	REGION 3 – Message preparation

	    IF NOT #iqUDT_FifoHeader.Status.Full       // FIFO isn't full
	    THEN
	        IF #ii_Gin <> #si_OldGin                // There is new GIN
	            AND NOT #sa_Status.InvalidGIN       // GIN is valid
	        THEN
	            REGION 3.1 - Sequencial ID
	                // ss_SequencialID character string clearing
	                #ss_SequencialID := '';
	                // ss_SequencialID integer input conversion to a character string
	                VAL_STRG(IN := "DB_GIN".GIN[#ii_Gin].FedEx.CustomerID,
	                         SIZE := 0,
	                         PREC := 0,
	                         FORMAT := 0,
	                         P := 1,
	                         OUT => #ss_SequencialID);
	                // Length of the ss_SequencialID character string
	                #si_StringLen := LEN(#ss_SequencialID);

	                // ss_SequencialID character string leading zeros addition
	                IF (#si_StringLen < 6)
	                THEN
	                    FOR #si_LenFillLoop := 1 TO 6 - #si_StringLen DO
	                        #ss_SequencialID := CONCAT(IN1 := '0',
	                                                   IN2 := #ss_SequencialID);
	                    END_FOR;
	                END_IF;
	            END_REGION

	            REGION 3.2 - LLC System ID
	                // Build LLC Syatem ID
	                #ss_LLCSystemID := CONCAT(IN1 := #is_DEPCOD,
	                                          IN2 := #is_LOConEquipment,
	                                          IN3 := #is_TYPofEquipment,
	                                          IN4 := #is_NumberOfTheEquipment);
	            END_REGION

	            REGION 3.3 - Package ID
	                // Build Package ID
	                #ss_PackageID := CONCAT(IN1 := #is_TrayCellNumber,
	                                        IN2 := #is_SorterNumber,
	                                        IN3 := #is_InductionNumber,
	                                        IN4 := #is_AreaNumber,
	                                        IN5 := #ss_SequencialID);
	            END_REGION

	            REGION 3.4 - Gap
	                // Gap character string clearing
	                #ss_Gap := '';
	                IF ("DB_GIN".GIN[#ii_Gin].General.LeadingGap > 999)
	                THEN
	                    #ss_Gap := '999';
	                ELSE
	                    // Gap integer input conversion to a character string
	                    VAL_STRG(IN := "DB_GIN".GIN[#ii_Gin].General.LeadingGap,
	                             SIZE := 0,
	                             PREC := 0,
	                             FORMAT := 0,
	                             P := 1,
	                             OUT => #ss_Gap);
	                    // Length of the gap character string
	                    #si_StringLen := LEN(#ss_Gap);
	                    // Gap character string leading zeros addition
	                    IF (#si_StringLen < 3)
	                    THEN
	                        FOR #si_LenFillLoop := 1 TO 3 - #si_StringLen DO
	                            #ss_Gap := CONCAT(IN1 := '0',
	                                              IN2 := #ss_Gap);
	                        END_FOR;

	                    END_IF;
	                END_IF;
	                #ss_GapUOM := 'CM';
	            END_REGION

	            REGION 3.5 – Message preparation
	                // Message composing according to the structure: STX,Body ,ETX
	                #ss_Message := CONCAT(IN1 := #cs_Start,
	                                      IN2 := #cs_Length,
	                                      IN3 := #cs_MessageType,
	                                      IN4 := #ss_LLCSystemID,
	                                      IN5 := #ss_PackageID,
	                                      IN6 := "DB_GIN".GIN[#ii_Gin].FedEx.HLCPackageID,
	                                      IN7 := #ss_Gap,
	                                      IN8 := #ss_GapUOM,
	                                      IN9 := #is_IncompatiblesUnit,
	                                      IN10 := "DB_GIN".GIN[#ii_Gin].FedEx.PalletType,
	                                      IN11 := "DB_GIN".GIN[#ii_Gin].FedEx.Mask,
	                                      IN12 := "DB_GIN".GIN[#ii_Gin].FedEx.CellNumber,
	                                      IN13 := "DB_GIN".GIN[#ii_Gin].FedEx.CellsOccupied,
	                                      IN14 := "DB_Time".Timestamp,
	                                      IN15 := #iUDT_Facility.TimeZoneDesignator,
	                                      IN16 := "DB_GIN".GIN[#ii_Gin].FedEx.BarcodeIdentification,
	                                      IN17 := "DB_GIN".GIN[#ii_Gin].FedEx.Barcodestatus,
	                                      IN18 := "DB_GIN".GIN[#ii_Gin].FedEx.Barcodedatalength,
	                                      IN19 := "DB_GIN".GIN[#ii_Gin].FedEx.Barcodedata,
	                                      IN20 := #cs_End);

	            END_REGION

	            REGION 3.6 – Maximum number of the message characters

	                #si_MaxMsgLen := "FC_GetNrOfArrayEl"(iv_Array := #sUDT_MessageArray.Character);

	            END_REGION

	            REGION 3.7 – Length of the complete message

	                #si_MsgLen := LEN(#ss_Message);

	                // Message length validation
	                #sa_Status.InvalidMessageLength := #si_MsgLen - 2 <> STRING_TO_INT(#cs_Length);

	            END_REGION

	            REGION 3.8 –  Message array size validation

	                #sa_Status.InvalidMsgArraySize := #si_MsgLen > #si_MaxMsgLen;

	            END_REGION

	            REGION 3.9 –  Message character string conversion to a message array of characters

	                IF (NOT #sa_Status.InvalidMsgArraySize)     // Message character array size is valid
	                THEN

	                    Strg_TO_Chars(Strg := #ss_Message,
	                                  pChars := 0,
	                                  Cnt => #sui_MsgArrayElNr,
	                                  Chars := #sUDT_MessageArray.Character);

	                END_IF;

	            END_REGION

	            REGION 3.10 – Clearing remaining characters in the message character array

	                IF (NOT #sa_Status.InvalidMsgArraySize)     // Message character array size is valid
	                THEN

	                    // Filling up not used message character array elements with '$00' (ASCII - 16#00)
	                    FILL_BLK(IN := #cc_NULL,
	                             COUNT := UINT_TO_ULINT(INT_TO_UINT(#si_MaxMsgLen) - #sui_MsgArrayElNr),
	                             OUT => #sUDT_MessageArray.Character[#sui_MsgArrayElNr]);

	                END_IF;

	            END_REGION

	            REGION 3.11 – Message write into a FIFO register

	                IF NOT #sa_Status.InvalidMsgArraySize           // Message character array size is valid
	                    AND NOT #sa_Status.InvalidMessageLength     //Message length is valid
	                THEN

	                    // Mode 'W' - Write FIFO record
	                    "FC_Fifo"(ic_Mode := 'W',
	                              qUDT_Status => #sa_Status.FIFOStatus,
	                              qx_Error => #sa_Status.FIFOError,
	                              qx_Warning => #sa_Status.FIFOWarning,
	                              iqv_Data := #sUDT_MessageArray,
	                              iqUDT_FifoHeader := #iqUDT_FifoHeader,
	                              iqv_DataBuffer := #iqa_FifoData);
	                ELSE
	                    #sa_Statistics.NotSentWrongMsgLen += 1;

	                END_IF;

	            END_REGION
	            #si_OldGin := #ii_Gin;
	        END_IF;

	        // In case of FIFO full, the FIFO full error bit and FIFO collective error bit are set
	    ELSE

	        #sa_Status.FIFOError := TRUE;
	        #sa_Status.FIFOStatus.FifoFull := TRUE;

	    END_IF;
	END_REGION

	REGION 4 - Writing outputs

	    #qx_Error := #sa_Status.InvalidMessageLength        // Invalid message length
	    OR #sa_Status.InvalidGIN                            // Invalid GIN
	    OR #sa_Status.InvalidMsgArraySize                   // Invalid message array size
	    OR #sa_Status.FIFOError;                            // FIFO error                                   // FIFO error

	END_REGION
END_FUNCTION_BLOCK

FUNCTION_BLOCK "FB_FedExLogInRequest"
TITLE = FB_Heartbeat
{ S7_Optimized_Access := 'TRUE' }
AUTHOR : MHSE
FAMILY : UPS_SpecificCommunication
VERSION : 3.0
// ATTRIBUTES
// AUTO_NUMBER = True
// BLOCK_NUMBER = 76
// END_ATTRIBUTES
//Function block to send and monitor the UPS heartbeat message.
   VAR_INPUT
      iUDT_Faciality { ExternalAccessible := 'False'; ExternalVisible := 'False'; ExternalWritable := 'False'} : "UDT_FedExFacility";   // System configuration
      ix_LogInRequest { ExternalAccessible := 'False'; ExternalVisible := 'False'; ExternalWritable := 'False'} : Bool;   // Log in message send request
   END_VAR

   VAR_OUTPUT
      qx_Error { ExternalAccessible := 'False'; ExternalVisible := 'False'; ExternalWritable := 'False'} : Bool;   // Collective error output
   END_VAR

   VAR_IN_OUT
      iqUDT_FifoHeader : "UDT_FifoHeader";   // FIFO header
      iqa_FifoData : Array[*] of "UDT_Message";   // FIFO data
      iqUDT_LoginStatus : "UDT_FedexLoginStatus";
   END_VAR

   VAR
      sR_TRIG_LogInRequest {InstructionName := 'R_TRIG'; LibVersion := '1.0'; ExternalAccessible := 'False'; ExternalVisible := 'False'; ExternalWritable := 'False'; S7_SetPoint := 'False'} : R_TRIG;   // Siemens "R_TRIG" - to prepare the rising edge trigger on "ix_LogInRequest" signal
      sUDT_MessageArray { ExternalAccessible := 'False'; ExternalVisible := 'False'; ExternalWritable := 'False'; S7_SetPoint := 'False'} : "UDT_Message";   // Message character array
      sa_Status { ExternalAccessible := 'False'; ExternalVisible := 'False'; ExternalWritable := 'False'} : Struct   // Status structure
         FIFOStatus { ExternalAccessible := 'False'; ExternalVisible := 'False'; ExternalWritable := 'False'} : "UDT_FifoStatus";   // FIFO status structure
         FIFOError { ExternalAccessible := 'False'; ExternalVisible := 'False'; ExternalWritable := 'False'; S7_SetPoint := 'True'} : Bool;   // FIFO data buffer full
         FIFOWarning { ExternalAccessible := 'False'; ExternalVisible := 'False'; ExternalWritable := 'False'; S7_SetPoint := 'True'} : Bool;   // FIFO error
         HeartbeatOk { ExternalAccessible := 'False'; ExternalVisible := 'False'; ExternalWritable := 'False'} : Bool;   // FIFO warning
         InvalidTimeInterval { ExternalAccessible := 'False'; ExternalVisible := 'False'; ExternalWritable := 'False'} : Bool;   // Heartbeat ok
         InvalidTimeout { ExternalAccessible := 'False'; ExternalVisible := 'False'; ExternalWritable := 'False'} : Bool;   // Heartbeat time interval lower than zero
         InvalidMsgArraySize { ExternalAccessible := 'False'; ExternalVisible := 'False'; ExternalWritable := 'False'} : Bool;   // Heartbeat timeout lower than zero or lower than heartbeat time interval
         InvalidSystemIDLen { ExternalAccessible := 'False'; ExternalVisible := 'False'; ExternalWritable := 'False'} : Bool;   //  Invalid designated system parameter input
         InvalidFacialityIDLen { ExternalAccessible := 'False'; ExternalVisible := 'False'; ExternalWritable := 'False'} : Bool;   //  Invalid GIN
      END_STRUCT;
      ss_Message { ExternalAccessible := 'False'; ExternalVisible := 'False'; ExternalWritable := 'False'} : String;   // Message character string
      sc_SS { ExternalAccessible := 'False'; ExternalVisible := 'False'; ExternalWritable := 'False'} : String;   // Maximum frequency of messages string
      ss_VersionID { ExternalAccessible := 'False'; ExternalVisible := 'False'; ExternalWritable := 'False'} : String;   // Version ID string
      sui_MsgArrayElNr { ExternalAccessible := 'False'; ExternalVisible := 'False'; ExternalWritable := 'False'} : UInt;   // Invalid message array size
      si_SSLen { ExternalAccessible := 'False'; ExternalVisible := 'False'; ExternalWritable := 'False'} : Int;   // Length of converted maximum frequency of messages string
      si_FacialityIDLen { ExternalAccessible := 'False'; ExternalVisible := 'False'; ExternalWritable := 'False'} : Int;   // Faciality ID length
      si_SystemIDLen { ExternalAccessible := 'False'; ExternalVisible := 'False'; ExternalWritable := 'False'} : Int;   // System ID length
      si_VersionIDLen { ExternalAccessible := 'False'; ExternalVisible := 'False'; ExternalWritable := 'False'} : Int;   // Version ID length
      si_MaxMsgLen { ExternalAccessible := 'False'; ExternalVisible := 'False'; ExternalWritable := 'False'} : Int;   // Maximum message length
      si_MsgLen { ExternalAccessible := 'False'; ExternalVisible := 'False'; ExternalWritable := 'False'} : Int;   // String character message length
      si_VersionIDLoop { ExternalAccessible := 'False'; ExternalVisible := 'False'; ExternalWritable := 'False'} : Int;   // Version ID spaces padding loop counter
   END_VAR

   VAR CONSTANT
      cc_NULL : Char := '$00';   // NULL sign
      cc_STX : Char := '$02';   // Start of the text
      cc_ETX : Char := '$03';   // End of the text
      cs_Length : String := '0035';   // Legth of the message
      cs_MessageType : String := 'LI';   // Message type
   END_VAR


BEGIN
	(*
	----------------------------------------------------------------------------------------

	Version history:
	Date        | Version   | Author        | Remark
	----------------------------------------------------------------------------------------
	29/06/2021  | 1.0       | F.Baten       | first release MHS TIA 16.0
	08/11/2021  | 1.1       | M.Piela       | Interface corrections
	05/04/2022  | 1.2       | K.Pokorski    | Review
	21/02/2023  | 4.0       | F.Baten       | 4.0 Release TIA 17.5
	*)

	REGION 1 – FIFO header status update

	    // Mode 'S' - FIFO register status update
	    "FC_Fifo"(ic_Mode := 'S',
	              qUDT_Status => #sa_Status.FIFOStatus,
	              qx_Error => #sa_Status.FIFOError,
	              qx_Warning => #sa_Status.FIFOWarning,
	              iqv_Data := #sUDT_MessageArray,
	              iqUDT_FifoHeader := #iqUDT_FifoHeader,
	              iqv_DataBuffer := #iqa_FifoData);


	END_REGION


	REGION 2 – Configuration check and create error

	    #si_FacialityIDLen := LEN(#iUDT_Faciality.FacilityID);
	    #si_SystemIDLen := LEN(#iUDT_Faciality.SystemID);

	    #sa_Status.InvalidSystemIDLen := #si_SystemIDLen <> 15;
	    #sa_Status.InvalidFacialityIDLen := #si_FacialityIDLen <> 6;

	END_REGION

	REGION 3 – Message preparation

	    #sR_TRIG_LogInRequest(CLK := #ix_LogInRequest);        // Log in request rising edge trigger detection

	    IF (NOT #iqUDT_FifoHeader.Status.Full)                 // FIFO isn't full
	    THEN

	        IF (NOT #sa_Status.FIFOError                                // No FIFO errors
	            AND NOT #sa_Status.InvalidSystemIDLen                   // Length of system ID field is ok
	            AND NOT #sa_Status.InvalidFacialityIDLen                // Length of faciality ID field is ok
	            AND #sR_TRIG_LogInRequest.Q)
	        THEN
	            REGION 3.1 – Message preparation

	                // Maximum frequency of messages to string conversion
	                #sc_SS := UDINT_TO_STRING(#iUDT_Faciality.SS);

	                // Delete "+"
	                #sc_SS := DELETE(IN := #sc_SS, L := 1, P := 1);

	                // Maximum frequency of messages length calculation
	                #si_SSLen := LEN(IN := #sc_SS);

	                // If maximum frequency of messages has only one digit then add leading zero
	                IF #si_SSLen = 1
	                THEN
	                    #sc_SS := CONCAT(IN1 := '0', IN2 := #sc_SS);

	                END_IF;

	                #ss_VersionID := #iUDT_Faciality.VersionID;

	                // Version ID length calculation
	                #si_VersionIDLen := LEN(#iUDT_Faciality.VersionID);

	                // IF Version ID length is less than 6, then padd it with spaces
	                IF #si_VersionIDLen < 6
	                THEN

	                    FOR #si_VersionIDLoop := 1 TO 6 - #si_VersionIDLen DO

	                        #ss_VersionID := CONCAT(IN1 := #ss_VersionID, IN2 := ' ');

	                    END_FOR;

	                END_IF;

	                // Heartbeat message composing according to the structure: STX,00,06,LS,ETX
	                #ss_Message := CONCAT(IN1 := #cc_STX,                       // Start of message
	                                      IN2 := #cs_Length,                    // Message length
	                                      IN3 := #cs_MessageType,               // Log-in request message
	                                      IN4 := #iUDT_Faciality.FacilityID,   // Generated during configuration. It is a fixed value for all systems
	                                      IN5 := #iUDT_Faciality.SystemID,     // System ID of the system making the request.
	                                      IN6 := #ss_VersionID,                 // Interface document version.
	                                      IN7 := #sc_SS,                        // Maximum ferquency of messages
	                                      IN8 := #cc_ETX);                      // End of message

	            END_REGION

	            REGION 3.2 – Maximum number of the message characters

	                #si_MaxMsgLen := "FC_GetNrOfArrayEl"(iv_Array := #sUDT_MessageArray.Character);

	            END_REGION

	            REGION 3.3 – Length of the complete message

	                #si_MsgLen := LEN(#ss_Message);

	            END_REGION

	            REGION 3.4 –  Message array size validation

	                #sa_Status.InvalidMsgArraySize := #si_MsgLen > #si_MaxMsgLen;

	            END_REGION

	            REGION 3.5 –  Message character string conversion to a message array of characters

	                IF (NOT #sa_Status.InvalidMsgArraySize)     // Message character array size is valid
	                THEN

	                    Strg_TO_Chars(Strg := #ss_Message,
	                                  pChars := 0,
	                                  Cnt => #sui_MsgArrayElNr,
	                                  Chars := #sUDT_MessageArray.Character);

	                END_IF;

	            END_REGION

	            REGION 3.6 – Clearing remaining characters in the message character array

	                IF (NOT #sa_Status.InvalidMsgArraySize)     // Message character array size is valid
	                THEN

	                    // Filling up not used message character array elements with '$00' (ASCII - 16#00)
	                    FILL_BLK(IN := #cc_NULL,
	                             COUNT := UINT_TO_ULINT(INT_TO_UINT(#si_MaxMsgLen) - #sui_MsgArrayElNr),
	                             OUT => #sUDT_MessageArray.Character[#sui_MsgArrayElNr]);

	                END_IF;

	            END_REGION

	            REGION 3.7 – Message write into a FIFO register

	                IF NOT #sa_Status.InvalidMsgArraySize // Message character array size is valid
	                THEN

	                    // Mode 'W' - Write FIFO record
	                    "FC_Fifo"(ic_Mode := 'W',
	                              qUDT_Status => #sa_Status.FIFOStatus,
	                              qx_Error => #sa_Status.FIFOError,
	                              qx_Warning => #sa_Status.FIFOWarning,
	                              iqv_Data := #sUDT_MessageArray,
	                              iqUDT_FifoHeader := #iqUDT_FifoHeader,
	                              iqv_DataBuffer := #iqa_FifoData);
	                END_IF;

	            END_REGION

	            #iqUDT_LoginStatus.Accepted := FALSE;
	            #iqUDT_LoginStatus.Rejected := FALSE;
	        END_IF;

	        // In case of FIFO full, the FIFO full error bit and FIFO collective error bit are set
	    ELSE

	        #sa_Status.FIFOError := TRUE;
	        #sa_Status.FIFOStatus.FifoFull := TRUE;

	    END_IF;

	END_REGION

	REGION 4 – Status

	    // Parametrization collective error output
	    #qx_Error :=
	    #sa_Status.InvalidSystemIDLen                               // Invalid System ID string length
	    OR #sa_Status.InvalidFacialityIDLen                         // Invalid Faciality ID lenght
	    OR #sa_Status.InvalidMsgArraySize                           // Invalid message array size
	    OR #sa_Status.FIFOError;                                    // FIFO error

	END_REGION
END_FUNCTION_BLOCK

FUNCTION_BLOCK "FB_FedExDecodeADC"
TITLE = FB_Decode
{ S7_Optimized_Access := 'TRUE' }
AUTHOR : MHSE
FAMILY : UPS_SpecificCommunication
VERSION : 3.0
// ATTRIBUTES
// AUTO_NUMBER = True
// BLOCK_NUMBER = 66
// END_ATTRIBUTES
//Function block to decode UPS messages.
   VAR_INPUT
      iUDT_FacilityADC { ExternalAccessible := 'False'; ExternalVisible := 'False'; ExternalWritable := 'False'} : "UDT_FedExFacility";   // ADC FedEx configuration
      ii_GinRangeStart { ExternalAccessible := 'False'; ExternalVisible := 'False'; ExternalWritable := 'False'} : Int;
      ii_GinRangeEnd { ExternalAccessible := 'False'; ExternalVisible := 'False'; ExternalWritable := 'False'} : Int;
      ii_UFORangeStart { ExternalAccessible := 'False'; ExternalVisible := 'False'; ExternalWritable := 'False'} : Int;
      ii_UFORangeEnd { ExternalAccessible := 'False'; ExternalVisible := 'False'; ExternalWritable := 'False'} : Int;
   END_VAR

   VAR_IN_OUT
      iqUDT_FifoRcvHeader : "UDT_FifoHeader";   // FIFO receive header
      iqv_FifoRcvData : Array[*] of "UDT_Message";   // FIFO receive data
      iqUDT_LoginStatus : "UDT_FedexLoginStatus";   // Login Status
      iqUDT_SI : Struct   // Buffer for SI message
         Data : "UDT_FedExMessageSI";   // SI message body
         NewMessage : Bool;   // New message received from ADC
      END_STRUCT;
      iqUDT_LR : Struct   // Buffer for LR message
         Data : "UDT_FedExMessageLoginResponse";   // LR message body
         NewMessage : Bool;   // New message received from ADC
      END_STRUCT;
      iqUDT_WS : Struct   // Buffer for WS message
         Data : "UDT_FedExMessageWS";   // WS message body
         NewMessage : Bool;   // New message received from ADC
      END_STRUCT;
      iqUDT_CustomerIDReference : "UDT_FedExCustomerID";
      iqx_UnexpectedDXReq { ExternalAccessible := 'False'; ExternalVisible := 'False'; ExternalWritable := 'False'} : Bool;   // Request DX message for GIN
      iqx_UnexpectedDLReq { ExternalAccessible := 'False'; ExternalVisible := 'False'; ExternalWritable := 'False'} : Bool;   // Request DL message for GIN
      iqx_HeartbeatOk { ExternalAccessible := 'False'; ExternalVisible := 'False'; ExternalWritable := 'False'} : Bool;   // Heartbeat signal was received
      iqx_ResetWritingTimer { ExternalAccessible := 'False'; ExternalVisible := 'False'; ExternalWritable := 'False'} : Bool;   // Reset writing timer in Heartbeat block
      iqx_ResetListeningTimer { ExternalAccessible := 'False'; ExternalVisible := 'False'; ExternalWritable := 'False'} : Bool;   // Reset listening timer in Heartbeat block
   END_VAR

   VAR
      sa_Status { ExternalAccessible := 'False'; ExternalVisible := 'False'; ExternalWritable := 'False'} : Struct   // Status structure
         BadMessage { ExternalAccessible := 'False'; ExternalVisible := 'False'; ExternalWritable := 'False'} : Array[1..10] of "UDT_Message";   //   Unknown message read
         FIFORcvStatus { ExternalAccessible := 'False'; ExternalVisible := 'False'; ExternalWritable := 'False'} : "UDT_FifoStatus";   //   Receive FIFO status structure
         FIFOError { ExternalAccessible := 'False'; ExternalVisible := 'False'; ExternalWritable := 'False'; S7_SetPoint := 'True'} : Bool;   //   FIFO error
         FIFOWarning { ExternalAccessible := 'False'; ExternalVisible := 'False'; ExternalWritable := 'False'; S7_SetPoint := 'True'} : Bool;   //   FIFO warning
         AcknowledgeError { ExternalAccessible := 'False'; ExternalVisible := 'False'; ExternalWritable := 'False'; S7_SetPoint := 'True'} : Bool;   //   Acknowledge error
         AcknowledgeWarning { ExternalAccessible := 'False'; ExternalVisible := 'False'; ExternalWritable := 'False'; S7_SetPoint := 'True'} : Bool;   //   Acknowledge warning
         HB_NotOK { ExternalAccessible := 'False'; ExternalVisible := 'False'; ExternalWritable := 'False'} : Bool;   //   Health bit not OK
      END_STRUCT;
      sUDT_FifoMsg { ExternalAccessible := 'False'; ExternalVisible := 'False'; ExternalWritable := 'False'; S7_SetPoint := 'False'} : "UDT_Message";   // Buffer for fifos message
      sUDT_MSGHeader { ExternalAccessible := 'False'; ExternalVisible := 'False'; ExternalWritable := 'False'; S7_SetPoint := 'False'} : "UDT_FedExMessageHeader";   // Read message header
      ss_NNNNNN { ExternalAccessible := 'False'; ExternalVisible := 'False'; ExternalWritable := 'False'} : String[6];   // Pacel GIN number of read message
      si_SizeOfMsg { ExternalAccessible := 'False'; ExternalVisible := 'False'; ExternalWritable := 'False'} : Int;   // Message array size
      si_GIN { ExternalAccessible := 'False'; ExternalVisible := 'False'; ExternalWritable := 'False'} : Int;   // Pacel GIN number of read message
      si_CustomerID { ExternalAccessible := 'False'; ExternalVisible := 'False'; ExternalWritable := 'False'} : Int;   // CustomerID of read message
      si_MessageLegth { ExternalAccessible := 'False'; ExternalVisible := 'False'; ExternalWritable := 'False'} : Int;   // Message length
      sx_InvalidLength { ExternalAccessible := 'False'; ExternalVisible := 'False'; ExternalWritable := 'False'} : Bool;   // Message invalid length
   END_VAR

   VAR_TEMP
      tx_MsgRead : Bool;   // Message read from FIFO
   END_VAR

   VAR CONSTANT
      cs_SI : String := 'SI';
      cs_WS : String := 'WS';
      cs_HB : String := 'HB';
      cs_LR : String := 'LR';
      cs_ConnectionAccepted : String := 'Y';
      ci_SizeSIMessage : Int := 388;
      ci_SizeWSMessage : Int := 92;
      ci_SizeLRMessage : Int := 66;
      ci_SizeHBMessage : Int := 6;
   END_VAR


BEGIN
	(*
	----------------------------------------------------------------------------------------

	Version history:
	Date        | Version   | Author        | Remark
	----------------------------------------------------------------------------------------
	01/11/2021  | 0.1       | N.Kadam       | first release MHS TIA 16
	05/04/2022  | 0.2       | K.Pokorski    | Review
	17.06.2022  | 0.3       | K. Pokorski   | Reset listening timer when any message is received
	07/07/2022  | 0.4       | K. Pokorski   | Reason code 3 issue fix in SI message
	21/02/2023  | 4.0       | F.Baten       | 4.0 Release TIA 17.5
	*)

	REGION 1 – FIFO header status update

	    // Mode 'S' - FIFO register status update
	    "FC_Fifo"(ic_Mode := 'S',
	              qUDT_Status => #sa_Status.FIFORcvStatus,
	              qx_Error => #sa_Status.FIFOError,
	              qx_Warning => #sa_Status.FIFOWarning,
	              iqv_Data := #sUDT_FifoMsg,
	              iqUDT_FifoHeader := #iqUDT_FifoRcvHeader,
	              iqv_DataBuffer := #iqv_FifoRcvData);

	    IF (NOT #iqUDT_FifoRcvHeader.Status.Empty                             // FIFO not empty
	        AND NOT #sa_Status.FIFOError)                                      // No FIFO error
	    THEN

	        // Mode 'R' - Read FIFO record
	        "FC_Fifo"(ic_Mode := 'R',
	                  qUDT_Status => #sa_Status.FIFORcvStatus,
	                  qx_Error => #sa_Status.FIFOError,
	                  qx_Warning => #sa_Status.FIFOWarning,
	                  iqv_Data := #sUDT_FifoMsg,
	                  iqUDT_FifoHeader := #iqUDT_FifoRcvHeader,
	                  iqv_DataBuffer := #iqv_FifoRcvData);

	        // Message read bit set and position initialize
	        #tx_MsgRead := TRUE;


	        // FIFO empty or FIFO error occured
	    ELSE

	        #tx_MsgRead := FALSE;

	    END_IF;

	END_REGION

	REGION 2 – Maximum number of the message characters

	    #si_SizeOfMsg := "FC_GetNrOfArrayEl"(iv_Array := #sUDT_FifoMsg.Character);

	END_REGION

	REGION 3 – Decoding header

	    IF #tx_MsgRead
	    THEN

	        "FC_FedExDecodeHeader"(iUDT_FifoMsg := #sUDT_FifoMsg,
	                               qUDT_MSGHeader => #sUDT_MSGHeader);

	    END_IF;
	END_REGION

	REGION 4 - Decode

	    IF #tx_MsgRead
	    THEN
	        #si_MessageLegth := STRING_TO_INT(#sUDT_MSGHeader.MessageLength);

	        IF
	            // Decode Login Response Message
	            #sUDT_MSGHeader.MessageType = #cs_LR
	        THEN
	            IF #si_MessageLegth = #ci_SizeLRMessage         // Check length of the message

	            THEN
	                Chars_TO_Strg(Chars := #sUDT_FifoMsg.Character,
	                              pChars := 7,
	                              Cnt := 6,
	                              Strg => #iqUDT_LR.Data.FacilityID);

	                Chars_TO_Strg(Chars := #sUDT_FifoMsg.Character,
	                              pChars := 13,
	                              Cnt := 15,
	                              Strg => #iqUDT_LR.Data.SystemID);

	                Chars_TO_Strg(Chars := #sUDT_FifoMsg.Character,
	                              pChars := 28,
	                              Cnt := 6,
	                              Strg => #iqUDT_LR.Data.VersionID);

	                Chars_TO_Strg(Chars := #sUDT_FifoMsg.Character,
	                              pChars := 34,
	                              Cnt := 1,
	                              Strg => #iqUDT_LR.Data.ConnectionStatus);

	                Chars_TO_Strg(Chars := #sUDT_FifoMsg.Character,
	                              pChars := 35,
	                              Cnt := 32,
	                              Strg => #iqUDT_LR.Data.LocalHost);

	                #iqx_ResetWritingTimer := TRUE;
	                #iqx_ResetListeningTimer := TRUE;
	                #iqUDT_LR.NewMessage := TRUE;

	                // Login Status verification  Y/N

	                IF #iqUDT_LR.Data.ConnectionStatus = #cs_ConnectionAccepted
	                    AND #iUDT_FacilityADC.FacilityID = #iqUDT_LR.Data.FacilityID
	                    AND #iUDT_FacilityADC.SystemID = #iqUDT_LR.Data.SystemID
	                    AND #iUDT_FacilityADC.VersionID = #iqUDT_LR.Data.VersionID
	                THEN
	                    #iqUDT_LoginStatus.Accepted := TRUE;    // Y = Accepted
	                    #iqUDT_LoginStatus.Rejected := FALSE;
	                ELSE
	                    #iqUDT_LoginStatus.Rejected := TRUE;   // N = Rejected
	                    #iqUDT_LoginStatus.Accepted := FALSE;
	                END_IF;
	            ELSE
	                #sx_InvalidLength := TRUE;
	                #iqUDT_LoginStatus.Rejected := TRUE;
	                #iqUDT_LoginStatus.Accepted := FALSE;
	            END_IF;

	        ELSIF

	            // //Decode Scan Information message
	            #sUDT_MSGHeader.MessageType = #cs_SI
	        THEN
	            IF #si_MessageLegth = #ci_SizeSIMessage
	            THEN
	                // Convert array of bytes into body structure.

	                Chars_TO_Strg(Chars := #sUDT_FifoMsg.Character,
	                              pChars := 7,
	                              Cnt := 15,
	                              Strg => #iqUDT_SI.Data.ADCSystemID);

	                Chars_TO_Strg(Chars := #sUDT_FifoMsg.Character,
	                              pChars := 22,
	                              Cnt := 1,
	                              Strg => #iqUDT_SI.Data.ScanUnitType);

	                Chars_TO_Strg(Chars := #sUDT_FifoMsg.Character,
	                              pChars := 23,
	                              Cnt := 6,
	                              Strg => #iqUDT_SI.Data.ImageID);

	                Chars_TO_Strg(Chars := #sUDT_FifoMsg.Character,
	                              pChars := 29,
	                              Cnt := 15,
	                              Strg => #iqUDT_SI.Data.PackageID);

	                Chars_TO_Strg(Chars := #sUDT_FifoMsg.Character,
	                              pChars := 44,
	                              Cnt := 10,
	                              Strg => #iqUDT_SI.Data.HLCPackageID);

	                Chars_TO_Strg(Chars := #sUDT_FifoMsg.Character,
	                              pChars := 54,
	                              Cnt := 15,
	                              Strg => #iqUDT_SI.Data.DIMSystemID);

	                Chars_TO_Strg(Chars := #sUDT_FifoMsg.Character,
	                              pChars := 69,
	                              Cnt := 5,
	                              Strg => #iqUDT_SI.Data.DimStatus);

	                Chars_TO_Strg(Chars := #sUDT_FifoMsg.Character,
	                              pChars := 74,
	                              Cnt := 6,
	                              Strg => #iqUDT_SI.Data.PackageDimLength);

	                Chars_TO_Strg(Chars := #sUDT_FifoMsg.Character,
	                              pChars := 80,
	                              Cnt := 6,
	                              Strg => #iqUDT_SI.Data.PackageDimWidth);

	                Chars_TO_Strg(Chars := #sUDT_FifoMsg.Character,
	                              pChars := 86,
	                              Cnt := 6,
	                              Strg => #iqUDT_SI.Data.PackageDimHeight);

	                Chars_TO_Strg(Chars := #sUDT_FifoMsg.Character,
	                              pChars := 92,
	                              Cnt := 2,
	                              Strg => #iqUDT_SI.Data.DIMUOM);

	                Chars_TO_Strg(Chars := #sUDT_FifoMsg.Character,
	                              pChars := 94,
	                              Cnt := 8,
	                              Strg => #iqUDT_SI.Data.DimLFTstatusCode);

	                Chars_TO_Strg(Chars := #sUDT_FifoMsg.Character,
	                              pChars := 102,
	                              Cnt := 25,
	                              Strg => #iqUDT_SI.Data.AlibiDims);

	                Chars_TO_Strg(Chars := #sUDT_FifoMsg.Character,
	                              pChars := 127,
	                              Cnt := 15,
	                              Strg => #iqUDT_SI.Data.SCLSystemID);

	                Chars_TO_Strg(Chars := #sUDT_FifoMsg.Character,
	                              pChars := 142,
	                              Cnt := 5,
	                              Strg => #iqUDT_SI.Data.SCLStatus);

	                Chars_TO_Strg(Chars := #sUDT_FifoMsg.Character,
	                              pChars := 147,
	                              Cnt := 6,
	                              Strg => #iqUDT_SI.Data.SCLWT);

	                Chars_TO_Strg(Chars := #sUDT_FifoMsg.Character,
	                              pChars := 153,
	                              Cnt := 2,
	                              Strg => #iqUDT_SI.Data.SCLWTUOM);

	                Chars_TO_Strg(Chars := #sUDT_FifoMsg.Character,
	                              pChars := 155,
	                              Cnt := 2,
	                              Strg => #iqUDT_SI.Data.SCLLFTStatusCode);

	                Chars_TO_Strg(Chars := #sUDT_FifoMsg.Character,
	                              pChars := 157,
	                              Cnt := 25,
	                              Strg => #iqUDT_SI.Data.AlibiWeight);

	                Chars_TO_Strg(Chars := #sUDT_FifoMsg.Character,
	                              pChars := 182,
	                              Cnt := 1,
	                              Strg => #iqUDT_SI.Data.Stackable);

	                Chars_TO_Strg(Chars := #sUDT_FifoMsg.Character,
	                              pChars := 183,
	                              Cnt := 17,
	                              Strg => #iqUDT_SI.Data.Timestamp);

	                Chars_TO_Strg(Chars := #sUDT_FifoMsg.Character,
	                              pChars := 200,
	                              Cnt := 5,
	                              Strg => #iqUDT_SI.Data.TimeZoneDesignator);

	                Chars_TO_Strg(Chars := #sUDT_FifoMsg.Character,
	                              pChars := 205,
	                              Cnt := 2,
	                              Strg => #iqUDT_SI.Data.CameraHeadstatus);

	                Chars_TO_Strg(Chars := #sUDT_FifoMsg.Character,
	                              pChars := 207,
	                              Cnt := 1,
	                              Strg => #iqUDT_SI.Data.PackageDataTruncated);

	                Chars_TO_Strg(Chars := #sUDT_FifoMsg.Character,
	                              pChars := 208,
	                              Cnt := 4,
	                              Strg => #iqUDT_SI.Data.TotalBarcodeDataLength);

	                Chars_TO_Strg(Chars := #sUDT_FifoMsg.Character,
	                              pChars := 212,
	                              Cnt := 3,
	                              Strg => #iqUDT_SI.Data.Barcode1Identification);

	                Chars_TO_Strg(Chars := #sUDT_FifoMsg.Character,
	                              pChars := 215,
	                              Cnt := 2,
	                              Strg => #iqUDT_SI.Data.Barcode1status);

	                Chars_TO_Strg(Chars := #sUDT_FifoMsg.Character,
	                              pChars := 217,
	                              Cnt := 4,
	                              Strg => #iqUDT_SI.Data.Barcode1datalength);

	                Chars_TO_Strg(Chars := #sUDT_FifoMsg.Character,
	                              pChars := 221,
	                              Cnt := 50,
	                              Strg => #iqUDT_SI.Data.Barcode1data);

	                Chars_TO_Strg(Chars := #sUDT_FifoMsg.Character,
	                              pChars := 271,
	                              Cnt := 3,
	                              Strg => #iqUDT_SI.Data.Barcode2Identification);

	                Chars_TO_Strg(Chars := #sUDT_FifoMsg.Character,
	                              pChars := 274,
	                              Cnt := 2,
	                              Strg => #iqUDT_SI.Data.Barcode2status);

	                Chars_TO_Strg(Chars := #sUDT_FifoMsg.Character,
	                              pChars := 276,
	                              Cnt := 4,
	                              Strg => #iqUDT_SI.Data.Barcode2datalength);

	                Chars_TO_Strg(Chars := #sUDT_FifoMsg.Character,
	                              pChars := 280,
	                              Cnt := 50,
	                              Strg => #iqUDT_SI.Data.Barcode2data);

	                Chars_TO_Strg(Chars := #sUDT_FifoMsg.Character,
	                              pChars := 330,
	                              Cnt := 3,
	                              Strg => #iqUDT_SI.Data.Barcode3Identification);

	                Chars_TO_Strg(Chars := #sUDT_FifoMsg.Character,
	                              pChars := 333,
	                              Cnt := 2,
	                              Strg => #iqUDT_SI.Data.Barcode3status);

	                Chars_TO_Strg(Chars := #sUDT_FifoMsg.Character,
	                              pChars := 335,
	                              Cnt := 4,
	                              Strg => #iqUDT_SI.Data.Barcode3datalength);

	                Chars_TO_Strg(Chars := #sUDT_FifoMsg.Character,
	                              pChars := 339,
	                              Cnt := 50,
	                              Strg => #iqUDT_SI.Data.Barcode3data);


	                // Message length is fixed and should be the same
	                IF #si_MessageLegth <> #ci_SizeSIMessage
	                THEN
	                    #sx_InvalidLength := TRUE;
	                ELSE
	                    #sx_InvalidLength := FALSE;
	                END_IF;
	                IF NOT #sx_InvalidLength
	                THEN
	                    // Convert 'NNNNNN' part in package ID to GIN number and store data in GIN database
	                    #ss_NNNNNN := RIGHT(IN := #iqUDT_SI.Data.PackageID, L := 6);
	                    STRG_VAL(IN := #ss_NNNNNN,
	                             FORMAT := 16#0,
	                             P := 1,
	                             OUT => #si_CustomerID);
	                    IF #si_CustomerID > 1 AND #si_CustomerID < 999999 THEN
	                        #si_GIN := #iqUDT_CustomerIDReference.CustomerIDReference[#si_CustomerID];
	                    END_IF;

	                    IF #si_GIN > 0
	                        AND #si_GIN < 9999 THEN

	                        // Generate SI message reason code
	                        IF "DB_GIN".GIN[#si_GIN].FedEx.PackageEntranceState = ' '
	                            OR ("DB_GIN".GIN[#si_GIN].FedEx.PackageEntranceState <> ' ' AND "DB_GIN".GIN[#si_GIN].FedEx.PackageExitState <> ' ')
	                            OR NOT ((#si_GIN >= #ii_GinRangeStart AND #si_GIN <= #ii_GinRangeEnd) OR (#si_GIN >= #ii_UFORangeStart AND #si_GIN <= #ii_UFORangeEnd))

	                        THEN
	                            "DB_GIN".GIN[#si_GIN].FedEx.ReasonCode := '3';

	                        ELSIF (#iqUDT_SI.Data.PackageDimLength = '      ' OR
	                            #iqUDT_SI.Data.PackageDimWidth = '      ' OR
	                            #iqUDT_SI.Data.PackageDimHeight = '      ')
	                            AND #iqUDT_SI.Data.DimStatus <> 'NOSYS' THEN
	                            "DB_GIN".GIN[#si_GIN].FedEx.ReasonCode := '2';

	                        ELSIF #iqUDT_SI.Data.SCLWT = '      '
	                            AND #iqUDT_SI.Data.SCLStatus <> 'NOSYS' THEN

	                            "DB_GIN".GIN[#si_GIN].FedEx.ReasonCode := '2';

	                        ELSIF "DB_GIN".GIN[#si_GIN].FedEx.ReasonCode = ' ' OR "DB_GIN".GIN[#si_GIN].FedEx.ReasonCode = '4' THEN
	                            "DB_GIN".GIN[#si_GIN].FedEx.ReasonCode := '0';

	                        ELSIF "DB_GIN".GIN[#si_GIN].FedEx.ReasonCode = '0' THEN
	                            "DB_GIN".GIN[#si_GIN].FedEx.ReasonCode := '5';


	                        END_IF;

	                        IF "DB_GIN".GIN[#si_GIN].FedEx.ReasonCode <> '3' THEN

	                            // Write data to DB_GIN
	                            "DB_GIN".GIN[#si_GIN].FedEx.ADCSystemID := #iqUDT_SI.Data.ADCSystemID;
	                            "DB_GIN".GIN[#si_GIN].FedEx.ScanUnitType := #iqUDT_SI.Data.ScanUnitType;
	                            "DB_GIN".GIN[#si_GIN].FedEx.ImageID := #iqUDT_SI.Data.ImageID;
	                            "DB_GIN".GIN[#si_GIN].FedEx.PackageID := #iqUDT_SI.Data.PackageID;
	                            "DB_GIN".GIN[#si_GIN].FedEx.HLCPackageID := #iqUDT_SI.Data.HLCPackageID;
	                            "DB_GIN".GIN[#si_GIN].FedEx.DIMSystemID := #iqUDT_SI.Data.DIMSystemID;
	                            "DB_GIN".GIN[#si_GIN].FedEx.DIMStatus := #iqUDT_SI.Data.DimStatus;
	                            "DB_GIN".GIN[#si_GIN].FedEx.PackageDimLength := #iqUDT_SI.Data.PackageDimLength;
	                            "DB_GIN".GIN[#si_GIN].FedEx.PackageDimWidth := #iqUDT_SI.Data.PackageDimWidth;
	                            "DB_GIN".GIN[#si_GIN].FedEx.PackageDimHeight := #iqUDT_SI.Data.PackageDimHeight;
	                            "DB_GIN".GIN[#si_GIN].FedEx.DIMUOM := #iqUDT_SI.Data.DIMUOM;
	                            "DB_GIN".GIN[#si_GIN].FedEx.DimLFTstatusCode := #iqUDT_SI.Data.DimLFTstatusCode;
	                            "DB_GIN".GIN[#si_GIN].FedEx.AlibiDims := #iqUDT_SI.Data.AlibiDims;
	                            "DB_GIN".GIN[#si_GIN].FedEx.SCLSystemID := #iqUDT_SI.Data.SCLSystemID;
	                            "DB_GIN".GIN[#si_GIN].FedEx.SCLStatus := #iqUDT_SI.Data.SCLStatus;
	                            "DB_GIN".GIN[#si_GIN].FedEx.SCLWT := #iqUDT_SI.Data.SCLWT;
	                            "DB_GIN".GIN[#si_GIN].FedEx.SCLWTUOM := #iqUDT_SI.Data.SCLWTUOM;
	                            "DB_GIN".GIN[#si_GIN].FedEx.SCLLFTStatusCode := #iqUDT_SI.Data.SCLLFTStatusCode;
	                            "DB_GIN".GIN[#si_GIN].FedEx.AlibiWeight := #iqUDT_SI.Data.AlibiWeight;
	                            "DB_GIN".GIN[#si_GIN].FedEx.Stackable := #iqUDT_SI.Data.Stackable;
	                            "DB_GIN".GIN[#si_GIN].FedEx.Stackable := #iqUDT_SI.Data.Timestamp;
	                            "DB_GIN".GIN[#si_GIN].FedEx.Stackable := #iqUDT_SI.Data.TimeZoneDesignator;
	                            "DB_GIN".GIN[#si_GIN].FedEx.CameraHeadstatus := #iqUDT_SI.Data.CameraHeadstatus;
	                            "DB_GIN".GIN[#si_GIN].FedEx.PackageDataTruncated := #iqUDT_SI.Data.PackageDataTruncated;
	                            "DB_GIN".GIN[#si_GIN].FedEx.TotalBarcodeDataLength := #iqUDT_SI.Data.TotalBarcodeDataLength;
	                            "DB_GIN".GIN[#si_GIN].FedEx.Barcode1Identification := #iqUDT_SI.Data.Barcode1Identification;
	                            "DB_GIN".GIN[#si_GIN].FedEx.Barcode1status := #iqUDT_SI.Data.Barcode1status;
	                            "DB_GIN".GIN[#si_GIN].FedEx.Barcode1datalength := #iqUDT_SI.Data.Barcode1datalength;
	                            "DB_GIN".GIN[#si_GIN].FedEx.Barcode1data := #iqUDT_SI.Data.Barcode1data;
	                            "DB_GIN".GIN[#si_GIN].FedEx.Barcode2Identification := #iqUDT_SI.Data.Barcode2Identification;
	                            "DB_GIN".GIN[#si_GIN].FedEx.Barcode2status := #iqUDT_SI.Data.Barcode2status;
	                            "DB_GIN".GIN[#si_GIN].FedEx.Barcode2datalength := #iqUDT_SI.Data.Barcode2datalength;
	                            "DB_GIN".GIN[#si_GIN].FedEx.Barcode2data := #iqUDT_SI.Data.Barcode2data;
	                            "DB_GIN".GIN[#si_GIN].FedEx.Barcode3Identification := #iqUDT_SI.Data.Barcode3Identification;
	                            "DB_GIN".GIN[#si_GIN].FedEx.Barcode3status := #iqUDT_SI.Data.Barcode3status;
	                            "DB_GIN".GIN[#si_GIN].FedEx.Barcode3datalength := #iqUDT_SI.Data.Barcode3datalength;
	                            "DB_GIN".GIN[#si_GIN].FedEx.Barcode3data := #iqUDT_SI.Data.Barcode3data;

	                        ELSE

	                            // Write data to DB_ExternalGIN when GIN is out of range
	                            "DB_ExternalGIN".UnexpectedSI.FedEx.ADCSystemID := #iqUDT_SI.Data.ADCSystemID;
	                            "DB_ExternalGIN".UnexpectedSI.FedEx.ScanUnitType := #iqUDT_SI.Data.ScanUnitType;
	                            "DB_ExternalGIN".UnexpectedSI.FedEx.ImageID := #iqUDT_SI.Data.ImageID;
	                            "DB_ExternalGIN".UnexpectedSI.FedEx.PackageID := #iqUDT_SI.Data.PackageID;
	                            "DB_ExternalGIN".UnexpectedSI.FedEx.HLCPackageID := #iqUDT_SI.Data.HLCPackageID;
	                            "DB_ExternalGIN".UnexpectedSI.FedEx.DIMSystemID := #iqUDT_SI.Data.DIMSystemID;
	                            "DB_ExternalGIN".UnexpectedSI.FedEx.DIMStatus := #iqUDT_SI.Data.DimStatus;
	                            "DB_ExternalGIN".UnexpectedSI.FedEx.PackageDimLength := #iqUDT_SI.Data.PackageDimLength;
	                            "DB_ExternalGIN".UnexpectedSI.FedEx.PackageDimWidth := #iqUDT_SI.Data.PackageDimWidth;
	                            "DB_ExternalGIN".UnexpectedSI.FedEx.PackageDimHeight := #iqUDT_SI.Data.PackageDimHeight;
	                            "DB_ExternalGIN".UnexpectedSI.FedEx.DIMUOM := #iqUDT_SI.Data.DIMUOM;
	                            "DB_ExternalGIN".UnexpectedSI.FedEx.DimLFTstatusCode := #iqUDT_SI.Data.DimLFTstatusCode;
	                            "DB_ExternalGIN".UnexpectedSI.FedEx.AlibiDims := #iqUDT_SI.Data.AlibiDims;
	                            "DB_ExternalGIN".UnexpectedSI.FedEx.SCLSystemID := #iqUDT_SI.Data.SCLSystemID;
	                            "DB_ExternalGIN".UnexpectedSI.FedEx.SCLStatus := #iqUDT_SI.Data.SCLStatus;
	                            "DB_ExternalGIN".UnexpectedSI.FedEx.SCLWT := #iqUDT_SI.Data.SCLWT;
	                            "DB_ExternalGIN".UnexpectedSI.FedEx.SCLWTUOM := #iqUDT_SI.Data.SCLWTUOM;
	                            "DB_ExternalGIN".UnexpectedSI.FedEx.SCLLFTStatusCode := #iqUDT_SI.Data.SCLLFTStatusCode;
	                            "DB_ExternalGIN".UnexpectedSI.FedEx.AlibiWeight := #iqUDT_SI.Data.AlibiWeight;
	                            "DB_ExternalGIN".UnexpectedSI.FedEx.Stackable := #iqUDT_SI.Data.Stackable;
	                            "DB_ExternalGIN".UnexpectedSI.FedEx.Stackable := #iqUDT_SI.Data.Timestamp;
	                            "DB_ExternalGIN".UnexpectedSI.FedEx.Stackable := #iqUDT_SI.Data.TimeZoneDesignator;
	                            "DB_ExternalGIN".UnexpectedSI.FedEx.CameraHeadstatus := #iqUDT_SI.Data.CameraHeadstatus;
	                            "DB_ExternalGIN".UnexpectedSI.FedEx.PackageDataTruncated := #iqUDT_SI.Data.PackageDataTruncated;
	                            "DB_ExternalGIN".UnexpectedSI.FedEx.TotalBarcodeDataLength := #iqUDT_SI.Data.TotalBarcodeDataLength;
	                            "DB_ExternalGIN".UnexpectedSI.FedEx.Barcode1Identification := #iqUDT_SI.Data.Barcode1Identification;
	                            "DB_ExternalGIN".UnexpectedSI.FedEx.Barcode1status := #iqUDT_SI.Data.Barcode1status;
	                            "DB_ExternalGIN".UnexpectedSI.FedEx.Barcode1datalength := #iqUDT_SI.Data.Barcode1datalength;
	                            "DB_ExternalGIN".UnexpectedSI.FedEx.Barcode1data := #iqUDT_SI.Data.Barcode1data;
	                            "DB_ExternalGIN".UnexpectedSI.FedEx.Barcode2Identification := #iqUDT_SI.Data.Barcode2Identification;
	                            "DB_ExternalGIN".UnexpectedSI.FedEx.Barcode2status := #iqUDT_SI.Data.Barcode2status;
	                            "DB_ExternalGIN".UnexpectedSI.FedEx.Barcode2datalength := #iqUDT_SI.Data.Barcode2datalength;
	                            "DB_ExternalGIN".UnexpectedSI.FedEx.Barcode2data := #iqUDT_SI.Data.Barcode2data;
	                            "DB_ExternalGIN".UnexpectedSI.FedEx.Barcode3Identification := #iqUDT_SI.Data.Barcode3Identification;
	                            "DB_ExternalGIN".UnexpectedSI.FedEx.Barcode3status := #iqUDT_SI.Data.Barcode3status;
	                            "DB_ExternalGIN".UnexpectedSI.FedEx.Barcode3datalength := #iqUDT_SI.Data.Barcode3datalength;
	                            "DB_ExternalGIN".UnexpectedSI.FedEx.Barcode3data := #iqUDT_SI.Data.Barcode3data;
	                            "DB_ExternalGIN".UnexpectedSI.FedEx.ReasonCode := '3';
	                            "DB_ExternalGIN".UnexpectedSI.FedEx.PackageID := #iqUDT_SI.Data.PackageID;
	                            "DB_ExternalGIN".UnexpectedSI.FedEx.CustomerID := #si_CustomerID;
	                            #iqx_UnexpectedDXReq := TRUE;// DX request
	                            #iqx_UnexpectedDLReq := TRUE;// DL request
	                        END_IF;




	                    END_IF;
	                    #iqx_ResetWritingTimer := TRUE;
	                    #iqx_ResetListeningTimer := TRUE;
	                    #iqUDT_SI.NewMessage := TRUE;
	                ELSE
	                    #sx_InvalidLength := TRUE;
	                END_IF;
	            END_IF;

	        ELSIF

	            //Decode Weight Scale Message
	            #sUDT_MSGHeader.MessageType = #cs_WS
	        THEN
	            IF #si_MessageLegth = #ci_SizeSIMessage
	            THEN
	                // Convert array of bytes into body structure.

	                Chars_TO_Strg(Chars := #sUDT_FifoMsg.Character,
	                              pChars := 7,
	                              Cnt := 15,
	                              Strg => #iqUDT_WS.Data.SCLSystemID);

	                Chars_TO_Strg(Chars := #sUDT_FifoMsg.Character,
	                              pChars := 22,
	                              Cnt := 15,
	                              Strg => #iqUDT_WS.Data.PackageID);

	                Chars_TO_Strg(Chars := #sUDT_FifoMsg.Character,
	                              pChars := 37,
	                              Cnt := 6,
	                              Strg => #iqUDT_WS.Data.SCLWT);

	                Chars_TO_Strg(Chars := #sUDT_FifoMsg.Character,
	                              pChars := 43,
	                              Cnt := 2,
	                              Strg => #iqUDT_WS.Data.SCLWTUOM);

	                Chars_TO_Strg(Chars := #sUDT_FifoMsg.Character,
	                              pChars := 45,
	                              Cnt := 2,
	                              Strg => #iqUDT_WS.Data.SCLLFTStatusCode);

	                Chars_TO_Strg(Chars := #sUDT_FifoMsg.Character,
	                              pChars := 47,
	                              Cnt := 25,
	                              Strg => #iqUDT_WS.Data.AlibiWeight);

	                Chars_TO_Strg(Chars := #sUDT_FifoMsg.Character,
	                              pChars := 72,
	                              Cnt := 17,
	                              Strg => #iqUDT_WS.Data.Timestamp);

	                Chars_TO_Strg(Chars := #sUDT_FifoMsg.Character,
	                              pChars := 89,
	                              Cnt := 5,
	                              Strg => #iqUDT_WS.Data.TimeZoneDesignator);



	                // Message length is fixed and should be the same
	                IF #si_MessageLegth <> #ci_SizeWSMessage
	                THEN
	                    #sx_InvalidLength := TRUE;
	                ELSE
	                    #sx_InvalidLength := FALSE;
	                END_IF;
	                IF NOT #sx_InvalidLength
	                THEN
	                    // Convert 'NNNNNN' part in package ID to GIN number and store data in GIN database
	                    #ss_NNNNNN := RIGHT(IN := #iqUDT_WS.Data.PackageID, L := 6);
	                    STRG_VAL(IN := #ss_NNNNNN,
	                             FORMAT := 16#0,
	                             P := 1,
	                             OUT => #si_CustomerID);

	                    IF #si_CustomerID > 1 AND #si_CustomerID < 999999 THEN
	                        #si_GIN := #iqUDT_CustomerIDReference.CustomerIDReference[#si_CustomerID];
	                    END_IF;

	                    "DB_GIN".GIN[#si_GIN].FedEx.SCLSystemID := #iqUDT_WS.Data.SCLSystemID;
	                    "DB_GIN".GIN[#si_GIN].FedEx.SCLSystemID := #iqUDT_WS.Data.PackageID;
	                    "DB_GIN".GIN[#si_GIN].FedEx.SCLWT := #iqUDT_WS.Data.SCLWT;
	                    "DB_GIN".GIN[#si_GIN].FedEx.SCLWTUOM := #iqUDT_WS.Data.SCLWTUOM;
	                    "DB_GIN".GIN[#si_GIN].FedEx.SCLLFTStatusCode := #iqUDT_WS.Data.SCLLFTStatusCode;
	                    "DB_GIN".GIN[#si_GIN].FedEx.AlibiWeight := #iqUDT_WS.Data.AlibiWeight;
	                    "DB_GIN".GIN[#si_GIN].FedEx.AlibiWeight := #iqUDT_WS.Data.Timestamp;
	                    "DB_GIN".GIN[#si_GIN].FedEx.AlibiWeight := #iqUDT_WS.Data.TimeZoneDesignator;

	                    #iqx_ResetWritingTimer := TRUE;
	                    #iqx_ResetListeningTimer := TRUE;
	                    #iqUDT_WS.NewMessage := TRUE;

	                ELSE
	                    #sx_InvalidLength := TRUE;

	                END_IF;
	            END_IF;

	        END_IF;


	    END_IF;
	END_REGION


	REGION 9 - Heartbeat Signal
	    // Message is read and type is HB
	    IF #tx_MsgRead
	        AND #sUDT_MSGHeader.MessageType = #cs_HB
	        AND #si_MessageLegth = #ci_SizeHBMessage
	    THEN
	        #iqx_HeartbeatOk := TRUE;

	    END_IF;
	END_REGION



END_FUNCTION_BLOCK

FUNCTION_BLOCK "FB_FedExLogOffRequest"
TITLE = FB_Heartbeat
{ S7_Optimized_Access := 'TRUE' }
AUTHOR : MHSE
FAMILY : UPS_SpecificCommunication
VERSION : 3.0
// ATTRIBUTES
// AUTO_NUMBER = True
// BLOCK_NUMBER = 78
// END_ATTRIBUTES
//Function block to send and monitor the UPS heartbeat message.
   VAR_INPUT
      i_UDT_Facility_PLC { ExternalAccessible := 'False'; ExternalVisible := 'False'; ExternalWritable := 'False'} : "UDT_FedExFacility";
      ix_LogOffRequest { ExternalAccessible := 'False'; ExternalVisible := 'False'; ExternalWritable := 'False'} : Bool;   // Log off message send request
      ix_Connected { ExternalAccessible := 'False'; ExternalVisible := 'False'; ExternalWritable := 'False'} : Bool;   // TCPIP connection established
      ix_ConnectionAccepted { ExternalAccessible := 'False'; ExternalVisible := 'False'; ExternalWritable := 'False'} : Bool;
   END_VAR

   VAR_OUTPUT
      qx_Error { ExternalAccessible := 'False'; ExternalVisible := 'False'; ExternalWritable := 'False'} : Bool;   // Error
   END_VAR

   VAR_IN_OUT
      iqUDT_FifoHeader : "UDT_FifoHeader";   // FIFO header
      iqa_FifoData : Array[*] of "UDT_Message";   // FIFO data
      iqx_Reconnect { ExternalAccessible := 'False'; ExternalVisible := 'False'; ExternalWritable := 'False'} : Bool;   // Re-establish connection
   END_VAR

